// TIA Portal project "Boiler_KVGM20" (V14)
// Программа управления котлом КВГМ-20

(* hardware
DEVICE "ET 200SP station_1"  ET 200SP-Station
   slot 0: "Rack_0"  Rack  6ES5 710-8MAx1
   slot 1: "PLC_1"  CPU 1510SP-1 PN  6ES7 510-1DJ01-0AB0  V2.1
   slot 2: "AI 8xI 2-,4-wire BA_1"  AI 8xI 2-,4-wire BA  6ES7 134-6GF00-0AA1  V1.0
      slot 1: "AI 8xI 2-,4-wire BA_1"  AI 8xI 2-,4-wire BA
   slot 3: "AI 8xI 2-,4-wire BA_2"  AI 8xI 2-,4-wire BA  6ES7 134-6GF00-0AA1  V1.0
      slot 1: "AI 8xI 2-,4-wire BA_2"  AI 8xI 2-,4-wire BA
   slot 4: "AI 8xI 2-,4-wire BA_3"  AI 8xI 2-,4-wire BA  6ES7 134-6GF00-0AA1  V1.0
      slot 1: "AI 8xI 2-,4-wire BA_3"  AI 8xI 2-,4-wire BA
   slot 5: "DI 16x24VDC ST_1"  DI 16x24VDC ST  6ES7 131-6BH00-0BA0  V1.1
      slot 1: "DI 16x24VDC ST_1"  DI 16x24VDC ST
   slot 6: "DI 16x24VDC ST_2"  DI 16x24VDC ST  6ES7 131-6BH00-0BA0  V1.1
      slot 1: "DI 16x24VDC ST_2"  DI 16x24VDC ST
   slot 7: "DI 16x24VDC ST_3"  DI 16x24VDC ST  6ES7 131-6BH00-0BA0  V1.1
      slot 1: "DI 16x24VDC ST_3"  DI 16x24VDC ST
   slot 8: "DI 16x24VDC ST_4"  DI 16x24VDC ST  6ES7 131-6BH00-0BA0  V1.1
      slot 1: "DI 16x24VDC ST_4"  DI 16x24VDC ST
   slot 9: "DI 16x24VDC ST_5"  DI 16x24VDC ST  6ES7 131-6BH00-0BA0  V1.1
      slot 1: "DI 16x24VDC ST_5"  DI 16x24VDC ST
   slot 10: "DI 16x24VDC ST_6"  DI 16x24VDC ST  6ES7 131-6BH00-0BA0  V1.1
      slot 1: "DI 16x24VDC ST_6"  DI 16x24VDC ST
   slot 11: "DQ 16x24VDC/0.5A ST_1"  DQ 16x24VDC/0.5A ST  6ES7 132-6BH00-0BA0  V1.1
      slot 1: "DQ 16x24VDC/0.5A ST_1"  DQ 16x24VDC/0.5A ST
   slot 12: "DQ 16x24VDC/0.5A ST_2"  DQ 16x24VDC/0.5A ST  6ES7 132-6BH00-0BA0  V1.1
      slot 1: "DQ 16x24VDC/0.5A ST_2"  DQ 16x24VDC/0.5A ST
   slot 13: "DQ 16x24VDC/0.5A ST_3"  DQ 16x24VDC/0.5A ST  6ES7 132-6BH00-0BA0  V1.1
      slot 1: "DQ 16x24VDC/0.5A ST_3"  DQ 16x24VDC/0.5A ST
   slot 14: "AQ 4xU/I ST_1"  AQ 4xU/I ST  6ES7 135-6HD00-0BA1  V1.1
      slot 1: "AQ 4xU/I ST_1"  AQ 4xU/I ST
   slot 15: "Server module_1"  Server module  6ES7 193-6PA00-0AA0  V1.1
      slot 1: "Server module_1"  Server module
   slot 127: "BA 2xRJ45"  BA 2xRJ45  6ES7 193-6AR00-0AA0  V0.0
      slot 32769: "Port_1"  6ES7 193-6AR00-0AA0
      slot 32770: "Port_2"  6ES7 193-6AR00-0AA0
*)

// ===== PLC "PLC_1"  CPU 1510SP-1 PN =====

VAR_GLOBAL   // PLC tag table "Default tag table"
   "Module1Chanel1" AT %IW0 : Int;
   "Module1Chanel2" AT %IW2 : Int;
   "Module1Chanel3" AT %IW4 : Int;
   "Module1Chanel4" AT %IW6 : Int;
   "Module1Chanel5" AT %IW8 : Int;
   "Module1Chanel6" AT %IW10 : Int;
   "Module1Chanel7" AT %IW12 : Int;
   "Module1Chanel8" AT %IW14 : Int;
   "Module2Chanel1" AT %IW16 : Int;
   "Module2Chanel2" AT %IW18 : Int;
   "Module2Chanel3" AT %IW20 : Int;
   "Module2Chanel4" AT %IW22 : Int;
   "Module2Chanel5" AT %IW24 : Int;
   "Module2Chanel6" AT %IW26 : Int;
   "Module2Chanel7" AT %IW28 : Int;
   "Module2Chanel8" AT %IW30 : Int;
   "Module3Chanel1" AT %IW32 : Int;
   "Module3Chanel2" AT %IW34 : Int;
   "Module3Chanel3" AT %IW36 : Int;
   "Module3Chanel4" AT %IW38 : Int;
   "Module3Chanel5" AT %IW40 : Int;
   "Module3Chanel6" AT %IW42 : Int;
   "Module3Chanel7" AT %IW44 : Int;
   "Module3Chanel8" AT %IW46 : Int;
   "Module4Chanel1" AT %I48.0 : Bool;
   "Module4Chanel2" AT %I48.1 : Bool;
   "Module4Chanel3" AT %I48.2 : Bool;
   "Module4Chanel4" AT %I48.3 : Bool;
   "Module4Chanel5" AT %I48.4 : Bool;
   "Module4Chanel6" AT %I48.5 : Bool;
   "Module4Chanel7" AT %I48.6 : Bool;
   "Module4Chanel8" AT %I48.7 : Bool;
   "Module4Chanel9" AT %I49.0 : Bool;
   "Module4Chanel10" AT %I49.1 : Bool;
   "Module4Chanel11" AT %I49.2 : Bool;
   "Module4Chanel12" AT %I49.3 : Bool;
   "Module4Chanel13" AT %I49.4 : Bool;
   "Module4Chanel14" AT %I49.5 : Bool;
   "Module4Chanel15" AT %I49.6 : Bool;
   "Module4Chanel16" AT %I49.7 : Bool;
   "Module5Chanel1" AT %I50.0 : Bool;
   "Module5Chanel2" AT %I50.1 : Bool;
   "Module5Chanel3" AT %I50.2 : Bool;
   "Module5Chanel4" AT %I50.3 : Bool;
   "Module5Chanel5" AT %I50.4 : Bool;
   "Module5Chanel6" AT %I50.5 : Bool;
   "Module5Chanel7" AT %I50.6 : Bool;
   "Module5Chanel8" AT %I50.7 : Bool;
   "Module5Chanel9" AT %I51.0 : Bool;
   "Module5Chanel10" AT %I51.1 : Bool;
   "Module5Chanel11" AT %I51.2 : Bool;
   "Module5Chanel12" AT %I51.3 : Bool;
   "Module5Chanel13" AT %I51.4 : Bool;
   "Module5Chanel14" AT %I51.5 : Bool;
   "Module5Chanel15" AT %I51.6 : Bool;
   "Module5Chanel16" AT %I51.7 : Bool;
   "Module6Chanel1" AT %I52.0 : Bool;
   "Module6Chanel2" AT %I52.1 : Bool;
   "Module6Chanel3" AT %I52.2 : Bool;
   "Module6Chanel4" AT %I52.3 : Bool;
   "Module6Chanel5" AT %I52.4 : Bool;
   "Module6Chanel6" AT %I52.5 : Bool;
   "Module6Chanel7" AT %I52.6 : Bool;
   "Module6Chanel8" AT %I52.7 : Bool;
   "Module6Chanel9" AT %I53.0 : Bool;
   "Module6Chanel10" AT %I53.1 : Bool;
   "Module6Chanel11" AT %I53.2 : Bool;
   "Module6Chanel12" AT %I53.3 : Bool;
   "Module6Chanel13" AT %I53.4 : Bool;
   "Module6Chanel14" AT %I53.5 : Bool;
   "Module6Chanel15" AT %I53.6 : Bool;
   "Module6Chanel16" AT %I53.7 : Bool;
   "Module7Chanel1" AT %I54.0 : Bool;
   "Module7Chanel2" AT %I54.1 : Bool;
   "Module7Chanel3" AT %I54.2 : Bool;
   "Module7Chanel4" AT %I54.3 : Bool;
   "Module7Chanel5" AT %I54.4 : Bool;
   "Module7Chanel6" AT %I54.5 : Bool;
   "Module7Chanel7" AT %I54.6 : Bool;
   "Module7Chanel8" AT %I54.7 : Bool;
   "Module7Chanel9" AT %I55.0 : Bool;
   "Module7Chanel10" AT %I55.1 : Bool;
   "Module7Chanel11" AT %I55.2 : Bool;
   "Module7Chanel12" AT %I55.3 : Bool;
   "Module7Chanel13" AT %I55.4 : Bool;
   "Module7Chanel14" AT %I55.5 : Bool;
   "Module7Chanel15" AT %I55.6 : Bool;
   "Module7Chanel16" AT %I55.7 : Bool;
   "Module8Chanel1" AT %I56.0 : Bool;
   "Module8Chanel2" AT %I56.1 : Bool;
   "Module8Chanel3" AT %I56.2 : Bool;
   "Module8Chanel4" AT %I56.3 : Bool;
   "Module8Chanel5" AT %I56.4 : Bool;
   "Module8Chanel6" AT %I56.5 : Bool;
   "Module8Chanel7" AT %I56.6 : Bool;
   "Module8Chanel8" AT %I56.7 : Bool;
   "Module8Chanel9" AT %I57.0 : Bool;
   "Module8Chanel10" AT %I57.1 : Bool;
   "Module8Chanel11" AT %I57.2 : Bool;
   "Module8Chanel12" AT %I57.3 : Bool;
   "Module8Chanel13" AT %I57.4 : Bool;
   "Module8Chanel14" AT %I57.5 : Bool;
   "Module8Chanel15" AT %I57.6 : Bool;
   "Module8Chanel16" AT %I57.7 : Bool;
   "Module9Chanel1" AT %I58.0 : Bool;
   "Module9Chanel2" AT %I58.1 : Bool;
   "Module9Chanel3" AT %I58.2 : Bool;
   "Module9Chanel4" AT %I58.3 : Bool;
   "Module9Chanel5" AT %I58.4 : Bool;
   "Module9Chanel6" AT %I58.5 : Bool;
   "Module9Chanel7" AT %I58.6 : Bool;
   "Module9Chanel8" AT %I58.7 : Bool;
   "Module9Chanel9" AT %I59.0 : Bool;
   "Module9Chanel10" AT %I59.1 : Bool;
   "Module9Chanel11" AT %I59.2 : Bool;
   "Module9Chanel12" AT %I59.3 : Bool;
   "Module9Chanel13" AT %I59.4 : Bool;
   "Module9Chanel14" AT %I59.5 : Bool;
   "Module9Chanel15" AT %I59.6 : Bool;
   "Module9Chanel16" AT %I59.7 : Bool;
   "Module10Chanel1" AT %Q0.0 : Bool;
   "Module10Chanel8" AT %Q0.7 : Bool;
   "Module10Chanel7" AT %Q0.6 : Bool;
   "Module10Chanel6" AT %Q0.5 : Bool;
   "Module10Chanel5" AT %Q0.4 : Bool;
   "Module10Chanel4" AT %Q0.3 : Bool;
   "Module10Chanel3" AT %Q0.2 : Bool;
   "Module10Chanel2" AT %Q0.1 : Bool;
   "Module10Chanel9" AT %Q1.0 : Bool;
   "Module10Chanel10" AT %Q1.1 : Bool;
   "Module10Chanel11" AT %Q1.2 : Bool;
   "Module10Chanel12" AT %Q1.3 : Bool;
   "Module10Chanel13" AT %Q1.4 : Bool;
   "Module10Chanel14" AT %Q1.5 : Bool;
   "Module10Chanel15" AT %Q1.6 : Bool;
   "Module10Chanel16" AT %Q1.7 : Bool;
   "Module11Chanel1" AT %Q2.0 : Bool;
   "Module11Chanel2" AT %Q2.1 : Bool;
   "Module11Chanel3" AT %Q2.2 : Bool;
   "Module11Chanel4" AT %Q2.3 : Bool;
   "Module11Chanel5" AT %Q2.4 : Bool;
   "Module11Chanel6" AT %Q2.5 : Bool;
   "Module11Chanel7" AT %Q2.6 : Bool;
   "Module11Chanel8" AT %Q2.7 : Bool;
   "Module11Chanel9" AT %Q3.0 : Bool;
   "Module11Chanel10" AT %Q3.1 : Bool;
   "Module11Chanel11" AT %Q3.2 : Bool;
   "Module11Chanel12" AT %Q3.3 : Bool;
   "Module11Chanel13" AT %Q3.4 : Bool;
   "Module11Chanel14" AT %Q3.5 : Bool;
   "Module11Chanel15" AT %Q3.6 : Bool;
   "Module11Chanel16" AT %Q3.7 : Bool;
   "Module12Chanel1" AT %Q4.0 : Bool;
   "Module12Chanel2" AT %Q4.1 : Bool;
   "Module12Chanel3" AT %Q4.2 : Bool;
   "Module12Chanel4" AT %Q4.3 : Bool;
   "Module12Chanel5" AT %Q4.4 : Bool;
   "Module12Chanel6" AT %Q4.5 : Bool;
   "Module12Chanel7" AT %Q4.6 : Bool;
   "Module12Chanel8" AT %Q4.7 : Bool;
   "Module12Chanel9" AT %Q5.0 : Bool;
   "Module12Chanel10" AT %Q5.1 : Bool;
   "Module12Chanel11" AT %Q5.2 : Bool;
   "Module12Chanel12" AT %Q5.3 : Bool;
   "Module12Chanel13" AT %Q5.4 : Bool;
   "Module12Chanel14" AT %Q5.5 : Bool;
   "Module12Chanel15" AT %Q5.6 : Bool;
   "Module12Chanel16" AT %Q5.7 : Bool;
   "Module13Chanel1" AT %QW6 : Int;
   "Module13Chanel2" AT %QW8 : Int;
   "Module13Chanel3" AT %QW10 : Int;
   "Module13Chanel4" AT %QW12 : Int;
   "FRONT_Btn_Ventilation_HMI" AT %M9.2 : Bool;   // Фронт нажатия кнопки ВЕНТИЛЯЦИЯ на HMI
   "FRONT_Btn_Ventilation_SCADA" AT %M9.3 : Bool;   // Фронт нажатия кнопки ВЕНТИЛЯЦИЯ на SCADA
   "FRONT_Btn_Ignition_HMI" AT %M9.4 : Bool;   // Фронт нажатия кнопки РОЗЖИГ на HMI
   "FRONT_Btn_Ignition_SCADA" AT %M9.5 : Bool;   // Фронт нажатия кнопки РОЗЖИГ на SCADA
   "FRONT_Btn_Normal_stop_HMI" AT %M9.6 : Bool;   // Фронт нажатия кнопки НОРМАЛЬНЫЙ ОСТАНОВ на HMI
   "FRONT_Btn_Normal_stop_SCADA" AT %M9.7 : Bool;   // Фронт нажатия кнопки НОРМАЛЬНЫЙ ОСТАНОВ на SCADA
   "FRONT_Btn_Alarm_stop_HMI" AT %M10.0 : Bool;   // Фронт нажатия кнопки АВАРИЙНЫЙ ОСТАНОВ на HMI
   "FRONT_Btn_Alarm_stop_SCADA" AT %M10.1 : Bool;   // Фронт нажатия кнопки АВАРИЙНЫЙ ОСТАНОВ на SCADA
   "FRONT_Btn_test_press_HMI" AT %M10.2 : Bool;   // Фронт нажатия кнопки ТЕСТОВАЯ ОПРЕССОВКА на HMI
   "FRONT_Btn_test_ignition_HMI" AT %M10.3 : Bool;   // Фронт нажатия кнопки ТЕСТОВЫЙ РОЗЖИГ на HMI
   "FRONT_Btn_manual_ignition_HMI" AT %M10.4 : Bool;   // Фронт нажатия кнопки РУЧНОЙ РОЗЖИГ на HMI
   "Gen_imp" AT %M10.5 : Bool;
   "FRONT_Alarm_1" AT %M10.6 : Bool;   // Фронт аварии1
   "FRONT_Alarm_2" AT %M10.7 : Bool;   // Фронт аварии2
   "FRONT_Alarm_3" AT %M11.0 : Bool;   // Фронт аварии3
   "FRONT_Alarm_4" AT %M11.1 : Bool;   // Фронт аварии4
   "FRONT_Alarm_5" AT %M11.2 : Bool;   // Фронт аварии5
   "FRONT_Alarm_6" AT %M11.3 : Bool;   // Фронт аварии6
   "FRONT_Alarm_7" AT %M11.4 : Bool;   // Фронт аварии7
   "FRONT_Alarm_8" AT %M11.5 : Bool;   // Фронт аварии8
   "FRONT_Alarm_9" AT %M11.6 : Bool;   // Фронт аварии9
   "FRONT_Alarm_10" AT %M11.7 : Bool;   // Фронт аварии10
   "FRONT_Alarm_11" AT %M12.0 : Bool;   // Фронт аварии11
   "FRONT_Alarm_12" AT %M12.1 : Bool;   // Фронт аварии12
   "FRONT_Alarm_13" AT %M12.2 : Bool;   // Фронт аварии13
   "FRONT_Alarm_14" AT %M12.3 : Bool;   // Фронт аварии14
   "FRONT_Alarm_15" AT %M12.4 : Bool;   // Фронт аварии15
   "FRONT_Alarm_16" AT %M12.5 : Bool;   // Фронт аварии16
   "FRONT_Alarm_17" AT %M12.6 : Bool;   // Фронт аварии17
   "FRONT_Btn_reset_sound_HMI" AT %M12.7 : Bool;   // Фронт нажатия кнопки СБРОС ЗВУКА на HMI
   "FRONT_DS_mode" AT %M13.0 : Bool;   // Фронт перевода ДС в ручной режим
   "FRONT_DV_mode" AT %M13.1 : Bool;   // Фронт перевода ДВ в ручной режим
   "FRONT_IVN_mode" AT %M13.2 : Bool;   // Фронт перевода ИВН в ручной режим
   "FRONT_KB_mode" AT %M13.3 : Bool;   // Фронт перевода КБ в ручной режим
   "FRONT_KO_mode" AT %M13.4 : Bool;   // Фронт перевода КО в ручной режим
   "FRONT_KZ_mode" AT %M13.5 : Bool;   // Фронт перевода КЗ в ручной режим
   "FRONT_PZK1_mode" AT %M13.6 : Bool;   // Фронт перевода ПЗК1 в ручной режим
   "FRONT_PZK2_mode" AT %M13.7 : Bool;   // Фронт перевода ПЗК2 в ручной режим
END_VAR

VAR_GLOBAL   // PLC tag table "www"
   "retval" AT %IW60 : Int;
END_VAR

TYPE "AI_sensor_4_20"
   STRUCT
      Enable : Bool;   // Наличие датчика
      N_module : USInt;   // № модуля (начиная с 1)
      N_chanel : USInt;   // № канала (начиная с 1)
      Value : Real;   // Текущее значение в физической величине
      Current_ADC : Int;   // Текущий код АЦП
      Low_limit_phisical_current : Real;   // Нижний предел датчика в физической величине текущий
      High_limit_phisical_current : Real := 100.0;   // Верхний предел датчика в физической величине текущий
      Low_limit_ADC_current : Int;   // Нижний предел датчика в АЦП текущий
      High_limit_ADC_current : Int := 27648;   // Верхний предел датчика в АЦП текущий
      Low_limit_phisical_new : Real;   // Нижний предел датчика в физической величине новый
      High_limit_phisical_new : Real := 100.0;   // Верхний предел датчика в физической величине новый
      Low_limit_ADC_new : Int;   // Нижний предел датчика в АЦП новый
      High_limit_ADC_new : Int := 27648;   // Верхний предел датчика в АЦП новый
      Apply : Bool;   // Применить
      Alarm_sensor : Bool;   // Неисправность датчика
      Current : Real;   // Текущее значение тока
      Reserv1 : Real;
      Reserv2 : Real;
      Reserv3 : Real;
      Reserv4 : Real;
   END_STRUCT;
END_TYPE

TYPE "DI_sensor"
   STRUCT
      Enable : Bool;   // Наличие датчика
      N_module : USInt;   // № модуля (начиная с 4)
      N_chanel : USInt;   // № канала (начиная с 1)
      Invert : Bool;   // Необходимость инвертирования сигнала
      Value : Bool;   // Текущее значение сигнала
      reserv1 : Bool;
      reserv2 : Bool;
   END_STRUCT;
END_TYPE

TYPE "DO_signal"
   STRUCT
      Enable : Bool;   // Наличие сигнала
      N_module : USInt;   // № модуля (начиная с 10)
      N_chanel : USInt;   // № канала (начиная с 1)
      Value : Bool;   // Текущее значение сигнала
      reserv1 : Bool;
      reserv2 : Bool;
   END_STRUCT;
END_TYPE

TYPE "AO_signal"
   STRUCT
      Enable : Bool;   // Наличие датчика
      N_module : USInt;   // № модуля (начиная с 13)
      N_chanel : USInt;   // № канала (начиная с 1)
      Value : Real;   // Текущее значение в физической величине
      Current_DAC : Int;   // Текущий код ЦАП
      Low_limit_phisical_current : Real;   // Нижний предел датчика в физической величине текущий
      High_limit_phisical_current : Real := 100.0;   // Верхний предел датчика в физической величине текущий
      Low_limit_phisical_new : Real;   // Нижний предел датчика в физической величине новый
      High_limit_phisical_new : Real := 100.0;   // Верхний предел датчика в физической величине новый
      Apply : Bool;   // Применить
      Reserv1 : Real;
      Reserv2 : Real;
      Reserv3 : Real;
      Reserv4 : Real;
   END_STRUCT;
END_TYPE

TYPE "Q_water"
   STRUCT
      Enable : Bool;   // Наличие параметра
      Value : Real;   // Значение
      "a" : Real := 0.6038;   // Коэффициент расхода
      Ksh : Real := 1.0;   // Поправочный коэффициент на шероховатость трубопровода
      Kp : Real := 1.00409;   // Поправочный коэффициент на неостроту входной кромки диафрагмы
      d : Real := 0.070696;   // Диаметр сужающего устройства
      ro : Real := 962.4729;   // Плотность среды в рабочих условиях
   END_STRUCT;
END_TYPE

TYPE "Q_gas"
   STRUCT
      Enable : Bool;   // Наличие параметра
      Value : Real;   // Значение
      "a" : Real := 0.60631;   // Коэффициент расхода
      Ksh : Real := 1.0;   // Поправочный коэффициент на шероховатость трубопровода
      Kp : Real := 1.00373;   // Поправочный коэффициент на неостроту входной кромки диафрагмы
      "E" : Real;   // Коэффициент расширения
      d : Real := 0.075498;   // Диаметр сужающего устройства
      ros : Real := 0.67245;   // Плотность среды в стандартных условиях
      Ps : Real := 101325.0;   // Давление в нормальных условиях
      Tgas : Real;   // Температура газа в рабочих условиях
      Tgas_fixed_value : Real;   // Температура газа в рабочих условиях фиксированное значение
      Tgas_fixed_value_on : Bool;   // Температура газа в рабочих условиях включить фиксированное значение
      K : Real := 0.99832;   // Коэффициент сжимаемости
      B4 : Real;   // Относительный диаметр сужающего устройства (в 4 степени)
      Dtrub : Real := 0.207;   // Диаметр трубопровода
      Pgas : Real;   // Давление газа в рабочих условиях
      Pgas_fixed_value : Real;   // Давление газа в рабочих условиях фиксированное значение
      Pgas_fixed_value_on : Bool;   // Давление газа в рабочих условиях включить фиксированное значение
   END_STRUCT;
END_TYPE

DATA_BLOCK "Sensors"   // DB1
{ S7_Optimized_Access := 'FALSE' }
VERSION : 0.1
   VAR
      T_water_before_boiler : "AI_sensor_4_20";   // Температура сетевой воды перед котлом (град С)
      P_water_before_boiler : "AI_sensor_4_20";   // Давление сетевой воды перед котлом (кгс/см2)
      dP_water_boiler : "AI_sensor_4_20";   // Перепад давления сетевой воды через котел (кПа)
      T_water_after_boiler : "AI_sensor_4_20";   // Температура сетевой воды после котла (град С)
      P_water_after_boiler : "AI_sensor_4_20";   // Давление сетевой воды после котла (кгс/см2)
      dP_water_boiler_1 : "AI_sensor_4_20";   // Перепад давления сетевой воды через котел (кПа)
      P_water_before_boiler_1 : "AI_sensor_4_20";   // Давление сетевой воды перед котлом (кгс/см2)
      dP_gas_boiler : "AI_sensor_4_20";   // Перепад давления газа на котел (кПа)
      dP_furnace_boiler : "AI_sensor_4_20";   // Разрежение в топке котла (Па)
      P_gas_before_PZK1_and_PZK2 : "AI_sensor_4_20";   // Давление газа между ПЗК-1 и ПЗК-2 (кПа)
      P_gas_before_burner : "AI_sensor_4_20";   // Давление газа перед горелкой (кПа)
      P_air_burner : "AI_sensor_4_20";   // Давление воздуха к горелке (Па)
      T_exhaust_gas : "AI_sensor_4_20";   // Температура уходящих газов (град С)
      ZRG_position : "AI_sensor_4_20";   // Положение рег. заслонки газа перед котлом (%)
      NAV_position : "AI_sensor_4_20";   // Положение направл. аппарата вентилятора (%)
      NAD_position : "AI_sensor_4_20";   // Положение направл. аппарата дымососа (%)
      DV_current_frequency : "AI_sensor_4_20";   // Текущ. значение ПЧ ДВ (Гц)
      DS_current_frequency : "AI_sensor_4_20";   // Текущ. значение ПЧ ДС (Гц)
      T_gas_before_BG : "AI_sensor_4_20";   // Температура газа перед БГ (град С)
      P_gas_before_BG : "AI_sensor_4_20";   // Давление газа перед БГ (кПа)
      Burner_flame : "DI_sensor";   // Наличие пламени горелки
      Igniter_flame : "DI_sensor";   // Наличие пламени запальника горелки
      KB_close : "DI_sensor";   // Клапан безопасности закрыт
      KO_open : "DI_sensor";   // Клапан опрессовки открыт
      KZ_open : "DI_sensor";   // Клапан запальника открыт
      PZK1_open : "DI_sensor";   // ПЗК-1 горелки открыт
      PZK2_not_close : "DI_sensor";   // ПЗК-2 горелки не закрыт
      P_gas_before_BG_min : "DI_sensor";   // Давление газа перед БГ мин.
      P_gas_before_BG_max : "DI_sensor";   // Давление газа перед БГ макс.
      P_air_before_burner_min : "DI_sensor";   // Давление воздуха перед горелкой мин.
      P_gas_before_burner_min : "DI_sensor";   // Давление газа перед горелкой мин.
      P_gas_before_burner_max : "DI_sensor";   // Давление газа перед горелкой макс.
      ZRG_open : "DI_sensor";   // Регулирующая заслонка газа. открыта
      ZRG_close : "DI_sensor";   // Регулирующая заслонка газа. закрыта
      ZRG_middle : "DI_sensor";   // Регулирующая заслонка газа. среднее
      ZRG_avto : "DI_sensor";   // Регулирующая заслонка газа. БРУ в положении "Авт"
      NAV_open : "DI_sensor";   // Регулирующая заслонка НАВ. открыта
      NAV_close : "DI_sensor";   // Регулирующая заслонка НАВ. закрыта
      NAV_middle : "DI_sensor";   // Регулирующая заслонка НАВ. среднее
      NAV_avto : "DI_sensor";   // Регулирующая заслонка НАВ. БРУ в положении "Авт"
      NAD_open : "DI_sensor";   // Регулирующая заслонка НАД. открыта
      NAD_close : "DI_sensor";   // Регулирующая заслонка НАД. закрыта
      NAD_middle : "DI_sensor";   // Регулирующая заслонка НАД. среднее
      NAD_avto : "DI_sensor";   // Регулирующая заслонка НАД. БРУ в положении "Авт"
      dP_furnace_boiler_min : "DI_sensor";   // Разрежение в топке котла мин.
      T_water_after_boiler_max : "DI_sensor";   // Температура сетевой воды после котла макс.
      Q_water_boiler_min : "DI_sensor";   // Расход сетевой воды через котел мин.
      Q_water_boiler_max : "DI_sensor";   // Расход сетевой воды через котел макс.
      P_water_after_boiler_min : "DI_sensor";   // Давление сетевой воды после котла мин.
      P_water_after_boiler_max : "DI_sensor";   // Давление сетевой воды после котла макс.
      P_water_before_boiler_min : "DI_sensor";   // Давление сетевой воды перед котлом мин.
      P_water_before_boiler_max : "DI_sensor";   // Давление сетевой воды перед котлом макс.
      Call_power_supply_сabinet : "DI_sensor";   // Вызов к шакафу электропитания
      DV_Invertor_alarm : "DI_sensor";   // Авария ПЧ ДВ
      DV_local_control : "DI_sensor";   // Управление «Местный» ДВ
      DV_dist_control : "DI_sensor";   // Управление «Дистанционный» ДВ
      DV_powergrid_mode : "DI_sensor";   // Режим "СЕТЬ" ДВ
      DV_invertor_mode : "DI_sensor";   // Режим "ПЧ" ДВ
      DV_invertor_QF_on : "DI_sensor";   // Автомат работы ДВ от ПЧ включен
      DV_powergrid_QF_on : "DI_sensor";   // Автомат работы ДВ от сети включен
      DV_invertor_on : "DI_sensor";   // Включен ДВ от ПЧ
      DV_powergrid_on : "DI_sensor";   // Включен ДВ от сети
      DV_no_voltage : "DI_sensor";   // Нет напряжения сети ШУД ДВ
      DS_Invertor_alarm : "DI_sensor";   // Авария ПЧ ДС
      DS_local_control : "DI_sensor";   // Управление «Местный» ДС
      DS_dist_control : "DI_sensor";   // Управление «Дистанционный» ДС
      DS_powergrid_mode : "DI_sensor";   // Режим "СЕТЬ" ДС
      DS_invertor_mode : "DI_sensor";   // Режим "ПЧ" ДС
      DS_invertor_QF_on : "DI_sensor";   // Автомат работы ДС от ПЧ включен
      DS_powergrid_QF_on : "DI_sensor";   // Автомат работы ДС от сети включен
      DS_invertor_on : "DI_sensor";   // ДС включен от ПЧ
      DS_powergrid_on : "DI_sensor";   // ДС включен от сети
      DS_no_voltage : "DI_sensor";   // Нет напряжения сети ШУД ДС
      CO_1 : "DI_sensor";   // Загазованность СО I порог
      CO_2 : "DI_sensor";   // Загазованность СО II порог
      CH4 : "DI_sensor";   // Загазованность CH4 порог
      Btn_STOP : "DI_sensor";   // Кнопка СТОП
      Btn_Ventilation : "DI_sensor";   // Кнопка Вентиляция
      Btn_Ignition : "DI_sensor";   // Кнопка Розжиг
      Btn_Sound : "DI_sensor";   // Кнопка Сброс звука / Проверка звука
      SHEU_voltage_ok : "DI_sensor";   // Контроль питания сети ~400В 1ШЭУ
      PZK2_open : "DI_sensor";   // ПЗК-2 горелки открыт
      Power_PLC_from_UPS : "DI_sensor";   // Питание контроллера от ИБП
      UPS_Low_charge : "DI_sensor";   // Заряд батареи ИБП низкий
      ZRG_voltage_ok : "DI_sensor";   // ЗРГ Напряжение в норме
      NAV_voltage_ok : "DI_sensor";   // НАВ Напряжение в норме
      NAD_voltage_ok : "DI_sensor";   // НАД Напряжение в норме
      ZDG_no_open : "DI_sensor";   // ЗДГ перед БГ. не открыта
      ZDG_no_close : "DI_sensor";   // ЗДГ перед БГ. не закрыта
      ZDG_opening : "DI_sensor";   // ЗДГ перед БГ. ход открытие
      ZDG_closing : "DI_sensor";   // ЗДГ перед БГ. ход закрытие
      ZDG_voltage_ok : "DI_sensor";   // ЗДГ перед БГ. Напряжение в норме
      ZDSV_before_boiler_no_open : "DI_sensor";   // ЗДСВ перед котлом. не открыта
      ZDSV_before_boiler_no_close : "DI_sensor";   // ЗДСВ перед котлом. не закрыта
      ZDSV_before_boiler_opening : "DI_sensor";   // ЗДСВ перед котлом. ход открытие
      ZDSV_before_boiler_closing : "DI_sensor";   // ЗДСВ перед котлом. ход закрытие
      ZDSV_before_boiler_voltage_ok : "DI_sensor";   // ЗДСВ перед котлом. Напряжение в норме
      ZDSV_before_boiler_limit_rotational_moment : "DI_sensor";   // ЗДСВ перед котлом. ограничитель крутящего момента
      ZDSV_after_boiler_no_open : "DI_sensor";   // ЗДСВ после котла. не открыта
      ZDSV_after_boiler_no_close : "DI_sensor";   // ЗДСВ после котла. не закрыта
      ZDSV_after_boiler_opening : "DI_sensor";   // ЗДСВ после котла. ход открытие
      ZDSV_after_boiler_closing : "DI_sensor";   // ЗДСВ после котла. ход закрытие
      ZDSV_after_boiler_voltage_ok : "DI_sensor";   // ЗДСВ после котла. Напряжение в норме
      ZDSV_after_boiler_limit_rotational_moment : "DI_sensor";   // ЗДСВ после котла. ограничитель крутящего момента
      ZRG_control_open : "DO_signal";   // ЗРГ команда «Больше»
      ZRG_control_close : "DO_signal";   // ЗРГ команда «Меньше»
      NAV_control_open : "DO_signal";   // НАВ команда «Больше»
      NAV_control_close : "DO_signal";   // НАВ команда «Меньше»
      NAD_control_open : "DO_signal";   // НАД команда «Больше»
      NAD_control_close : "DO_signal";   // НАД команда «Меньше»
      Indication_RUN : "DO_signal";   // Индикация «Работа»
      Indication_ALARM : "DO_signal";   // Индикация «Авария»
      Indication_NORMA : "DO_signal";   // Индикация «Защиты в норме»
      Indication_READY : "DO_signal";   // Индикация «Готов к розжигу»
      ZDG_control_open : "DO_signal";   // ЗДГ команда «открыть»
      ZDG_control_close : "DO_signal";   // ЗДГ команда «закрыть»
      ZDG_control_stop : "DO_signal";   // ЗДГ команда «стоп»
      ZDG_control_disable_open : "DO_signal";   // ЗДГ команда «запрет открытия»
      KB_control_close : "DO_signal";   // КБ команда «закрыть»
      KO_control_open : "DO_signal";   // КО команда «открыть»
      KZ_control_open : "DO_signal";   // КЗ команда «открыть»
      IVN_control_on : "DO_signal";   // ИВН команда «включить»
      PZK1_control_open : "DO_signal";   // ПЗК1 команда «открыть»
      PZK2_control_open : "DO_signal";   // ПЗК2 команда «открыть»
      ZDSV_before_boiler_control_open : "DO_signal";   // ЗДСВ перед котлом команда «открыть»
      ZDSV_before_boiler_control_close : "DO_signal";   // ЗДСВ перед котлом команда «закрыть»
      ZDSV_before_boiler_control_stop : "DO_signal";   // ЗДСВ перед котлом команда «стоп»
      ZDSV_before_boiler_control_disable_close : "DO_signal";   // ЗДСВ перед котлом команда «запрет закрытия»
      ZDSV_after_boiler_control_open : "DO_signal";   // ЗДСВ после котла команда «открыть»
      ZDSV_after_boiler_control_close : "DO_signal";   // ЗДСВ после котла команда «закрыть»
      ZDSV_after_boiler_control_stop : "DO_signal";   // ЗДСВ после котла команда «стоп»
      ZDSV_after_boiler_control_disable_close : "DO_signal";   // ЗДСВ после котла команда «запрет закрытия»
      control_alarm_signal : "DO_signal";   // Включение аварийной сигнализации
      DV_control_start : "DO_signal";   // ДВ команда «пуск»
      DV_control_stop : "DO_signal";   // ДВ команда «стоп»
      DS_control_start : "DO_signal";   // ДС команда «пуск»
      DS_control_stop : "DO_signal";   // ДС команда «стоп»
      DV_control_frequency : "AO_signal";   // Задание для ПЧ ДВ
      DS_control_frequency : "AO_signal";   // Задание для ПЧ ДС
      Q_water_boiler : "Q_water";   // Расход сетевой воды через котел (м3/ч)
      Q_gas : "Q_gas";   // Расход газа (м3/ч)
   END_VAR
BEGIN
   T_water_before_boiler.Enable := true;
   T_water_before_boiler.N_module := 1;
   T_water_before_boiler.N_chanel := 1;
   P_water_before_boiler.Enable := true;
   dP_water_boiler.Enable := true;
   T_water_after_boiler.Enable := true;
   P_water_after_boiler.Enable := true;
   dP_water_boiler_1.Enable := true;
   P_water_before_boiler_1.Enable := true;
   dP_gas_boiler.Enable := true;
   dP_furnace_boiler.Enable := true;
   P_gas_before_PZK1_and_PZK2.Enable := true;
   P_gas_before_burner.Enable := true;
   P_air_burner.Enable := true;
   T_exhaust_gas.Enable := true;
   ZRG_position.Enable := true;
   NAV_position.Enable := true;
   NAD_position.Enable := true;
   DV_current_frequency.Enable := true;
   DS_current_frequency.Enable := true;
   P_water_before_boiler.N_module := 1;
   P_water_before_boiler.N_chanel := 2;
   dP_water_boiler.N_module := 1;
   dP_water_boiler.N_chanel := 3;
   T_water_after_boiler.N_module := 1;
   T_water_after_boiler.N_chanel := 4;
   P_water_after_boiler.N_module := 1;
   P_water_after_boiler.N_chanel := 5;
   dP_water_boiler_1.N_module := 1;
   dP_water_boiler_1.N_chanel := 6;
   P_water_before_boiler_1.N_module := 1;
   P_water_before_boiler_1.N_chanel := 7;
   dP_gas_boiler.N_module := 1;
   dP_gas_boiler.N_chanel := 8;
   dP_furnace_boiler.N_module := 2;
   dP_furnace_boiler.N_chanel := 1;
   P_gas_before_PZK1_and_PZK2.N_module := 2;
   P_gas_before_PZK1_and_PZK2.N_chanel := 2;
   P_gas_before_burner.N_module := 2;
   P_gas_before_burner.N_chanel := 3;
   P_air_burner.N_module := 2;
   P_air_burner.N_chanel := 4;
   T_exhaust_gas.N_module := 2;
   T_exhaust_gas.N_chanel := 5;
   ZRG_position.N_module := 2;
   ZRG_position.N_chanel := 6;
   NAV_position.N_module := 2;
   NAV_position.N_chanel := 7;
   NAD_position.N_module := 2;
   NAD_position.N_chanel := 8;
   DV_current_frequency.N_module := 3;
   DV_current_frequency.N_chanel := 1;
   DS_current_frequency.N_module := 3;
   DS_current_frequency.N_chanel := 2;
   T_water_before_boiler.Low_limit_phisical_current := 0.0;
   T_water_before_boiler.High_limit_phisical_current := 200.0;
   T_water_before_boiler.Low_limit_phisical_new := 0.0;
   T_water_before_boiler.High_limit_phisical_new := 200.0;
   dP_gas_boiler.High_limit_phisical_current := 16.0;
   dP_gas_boiler.High_limit_phisical_new := 16.0;
   P_gas_before_PZK1_and_PZK2.High_limit_phisical_current := 40.0;
   P_gas_before_PZK1_and_PZK2.High_limit_phisical_new := 40.0;
   P_gas_before_burner.High_limit_phisical_current := 40.0;
   P_gas_before_burner.High_limit_phisical_new := 40.0;
   dP_furnace_boiler.Low_limit_phisical_current := -200.0;
   dP_furnace_boiler.High_limit_phisical_current := 200.0;
   dP_furnace_boiler.Low_limit_phisical_new := -200.0;
   dP_furnace_boiler.High_limit_phisical_new := 200.0;
   T_exhaust_gas.High_limit_phisical_current := 300.0;
   T_exhaust_gas.High_limit_phisical_new := 300.0;
   P_air_burner.High_limit_phisical_current := 2500.0;
   P_air_burner.High_limit_phisical_new := 2500.0;
   T_water_after_boiler.High_limit_phisical_current := 200.0;
   T_water_after_boiler.High_limit_phisical_new := 200.0;
   P_water_before_boiler.High_limit_phisical_current := 160.0;
   P_water_before_boiler.High_limit_phisical_new := 160.0;
   dP_water_boiler.High_limit_phisical_current := 400.0;
   dP_water_boiler.High_limit_phisical_new := 400.0;
   P_water_after_boiler.High_limit_phisical_current := 16.0;
   P_water_after_boiler.High_limit_phisical_new := 16.0;
   dP_water_boiler_1.High_limit_phisical_current := 400.0;
   dP_water_boiler_1.High_limit_phisical_new := 400.0;
   P_water_before_boiler_1.High_limit_phisical_new := 16.0;
   P_water_before_boiler_1.High_limit_phisical_current := 16.0;
   DV_current_frequency.High_limit_phisical_current := 50.0;
   DV_current_frequency.High_limit_phisical_new := 50.0;
   DS_current_frequency.High_limit_phisical_current := 50.0;
   DS_current_frequency.High_limit_phisical_new := 50.0;
   T_gas_before_BG.High_limit_phisical_current := 200.0;
   T_gas_before_BG.High_limit_phisical_new := 200.0;
   P_gas_before_BG.High_limit_phisical_current := 40.0;
   P_gas_before_BG.High_limit_phisical_new := 40.0;
   Burner_flame.Enable := true;
   Igniter_flame.Enable := true;
   KB_close.Enable := true;
   KO_open.Enable := true;
   KZ_open.Enable := true;
   PZK1_open.Enable := true;
   PZK2_not_close.Enable := true;
   P_gas_before_BG_min.Enable := true;
   P_gas_before_BG_max.Enable := true;
   P_air_before_burner_min.Enable := true;
   P_gas_before_burner_min.Enable := true;
   P_gas_before_burner_max.Enable := true;
   ZRG_open.Enable := true;
   ZRG_close.Enable := true;
   ZRG_middle.Enable := true;
   ZRG_avto.Enable := true;
   NAV_open.Enable := true;
   NAV_close.Enable := true;
   NAV_middle.Enable := true;
   NAV_avto.Enable := true;
   NAD_open.Enable := true;
   NAD_close.Enable := true;
   NAD_middle.Enable := true;
   NAD_avto.Enable := true;
   dP_furnace_boiler_min.Enable := true;
   T_water_after_boiler_max.Enable := true;
   Q_water_boiler_min.Enable := true;
   Q_water_boiler_max.Enable := true;
   P_water_after_boiler_min.Enable := true;
   P_water_after_boiler_max.Enable := true;
   P_water_before_boiler_min.Enable := true;
   P_water_before_boiler_max.Enable := true;
   Call_power_supply_сabinet.Enable := true;
   DV_Invertor_alarm.Enable := true;
   DV_local_control.Enable := true;
   DV_dist_control.Enable := true;
   DV_powergrid_mode.Enable := true;
   DV_invertor_mode.Enable := true;
   DV_invertor_QF_on.Enable := true;
   DV_powergrid_QF_on.Enable := true;
   DV_invertor_on.Enable := true;
   DV_powergrid_on.Enable := true;
   DV_no_voltage.Enable := true;
   DS_Invertor_alarm.Enable := true;
   DS_local_control.Enable := true;
   DS_dist_control.Enable := true;
   DS_powergrid_mode.Enable := true;
   DS_invertor_mode.Enable := true;
   DS_invertor_QF_on.Enable := true;
   DS_powergrid_QF_on.Enable := true;
   DS_invertor_on.Enable := true;
   DS_powergrid_on.Enable := true;
   DS_no_voltage.Enable := true;
   CO_1.Enable := true;
   CO_2.Enable := true;
   CH4.Enable := true;
   SHEU_voltage_ok.Enable := true;
   PZK2_open.Enable := true;
   Power_PLC_from_UPS.Enable := true;
   ZRG_voltage_ok.Enable := true;
   NAV_voltage_ok.Enable := true;
   NAD_voltage_ok.Enable := true;
   ZDG_no_open.Enable := true;
   ZDG_no_close.Enable := true;
   ZDG_opening.Enable := true;
   ZDG_closing.Enable := true;
   ZDG_voltage_ok.Enable := true;
   ZDSV_before_boiler_no_open.Enable := true;
   ZDSV_before_boiler_no_close.Enable := true;
   ZDSV_before_boiler_opening.Enable := true;
   ZDSV_before_boiler_closing.Enable := true;
   ZDSV_before_boiler_voltage_ok.Enable := true;
   ZDSV_before_boiler_limit_rotational_moment.Enable := true;
   ZDSV_after_boiler_no_open.Enable := true;
   ZDSV_after_boiler_no_close.Enable := true;
   ZDSV_after_boiler_opening.Enable := true;
   ZDSV_after_boiler_closing.Enable := true;
   ZDSV_after_boiler_voltage_ok.Enable := true;
   ZDSV_after_boiler_limit_rotational_moment.Enable := true;
   Burner_flame.N_module := 4;
   Burner_flame.N_chanel := 1;
   Igniter_flame.N_module := 4;
   Igniter_flame.N_chanel := 2;
   KB_close.N_module := 4;
   KB_close.N_chanel := 3;
   KO_open.N_module := 4;
   KO_open.N_chanel := 4;
   KZ_open.N_module := 4;
   KZ_open.N_chanel := 5;
   PZK1_open.N_module := 4;
   PZK1_open.N_chanel := 6;
   PZK2_not_close.N_module := 4;
   PZK2_not_close.N_chanel := 7;
   P_gas_before_BG_min.N_module := 4;
   P_gas_before_BG_min.N_chanel := 8;
   P_gas_before_BG_max.N_module := 4;
   P_gas_before_BG_max.N_chanel := 9;
   P_air_before_burner_min.N_module := 4;
   P_air_before_burner_min.N_chanel := 10;
   P_gas_before_burner_min.N_module := 4;
   P_gas_before_burner_min.N_chanel := 11;
   P_gas_before_burner_max.N_module := 4;
   P_gas_before_burner_max.N_chanel := 12;
   ZRG_open.N_module := 4;
   ZRG_open.N_chanel := 13;
   ZRG_close.N_module := 4;
   ZRG_close.N_chanel := 14;
   ZRG_middle.N_module := 4;
   ZRG_middle.N_chanel := 15;
   ZRG_avto.N_module := 4;
   ZRG_avto.N_chanel := 16;
   NAV_open.N_module := 5;
   NAV_open.N_chanel := 1;
   NAV_close.N_module := 5;
   NAV_close.N_chanel := 2;
   NAV_middle.N_module := 5;
   NAV_middle.N_chanel := 3;
   NAV_avto.N_module := 5;
   NAV_avto.N_chanel := 4;
   NAD_open.N_module := 5;
   NAD_open.N_chanel := 5;
   NAD_close.N_module := 5;
   NAD_close.N_chanel := 6;
   NAD_middle.N_module := 5;
   NAD_middle.N_chanel := 7;
   NAD_avto.N_module := 5;
   NAD_avto.N_chanel := 8;
   dP_furnace_boiler_min.N_module := 5;
   dP_furnace_boiler_min.N_chanel := 9;
   T_water_after_boiler_max.N_module := 5;
   T_water_after_boiler_max.N_chanel := 10;
   Q_water_boiler_min.N_module := 5;
   Q_water_boiler_min.N_chanel := 11;
   Q_water_boiler_max.N_module := 5;
   Q_water_boiler_max.N_chanel := 12;
   P_water_after_boiler_min.N_module := 5;
   P_water_after_boiler_min.N_chanel := 13;
   P_water_after_boiler_max.N_module := 5;
   P_water_after_boiler_max.N_chanel := 14;
   P_water_before_boiler_min.N_module := 5;
   P_water_before_boiler_min.N_chanel := 15;
   P_water_before_boiler_max.N_module := 5;
   P_water_before_boiler_max.N_chanel := 16;
   Call_power_supply_сabinet.N_module := 6;
   Call_power_supply_сabinet.N_chanel := 1;
   DV_Invertor_alarm.N_module := 6;
   DV_Invertor_alarm.N_chanel := 2;
   DV_local_control.N_module := 6;
   DV_local_control.N_chanel := 3;
   DV_dist_control.N_module := 6;
   DV_dist_control.N_chanel := 4;
   DV_powergrid_mode.N_module := 6;
   DV_powergrid_mode.N_chanel := 5;
   DV_invertor_mode.N_module := 6;
   DV_invertor_mode.N_chanel := 6;
   DV_invertor_QF_on.N_module := 6;
   DV_invertor_QF_on.N_chanel := 7;
   DV_powergrid_QF_on.N_module := 6;
   DV_powergrid_QF_on.N_chanel := 8;
   DV_invertor_on.N_module := 6;
   DV_invertor_on.N_chanel := 9;
   DV_powergrid_on.N_module := 6;
   DV_powergrid_on.N_chanel := 10;
   DV_no_voltage.N_module := 6;
   DV_no_voltage.N_chanel := 11;
   DS_Invertor_alarm.N_module := 6;
   DS_Invertor_alarm.N_chanel := 12;
   DS_local_control.N_module := 6;
   DS_local_control.N_chanel := 13;
   DS_dist_control.N_module := 6;
   DS_dist_control.N_chanel := 14;
   DS_powergrid_mode.N_module := 6;
   DS_powergrid_mode.N_chanel := 15;
   DS_invertor_mode.N_module := 6;
   DS_invertor_mode.N_chanel := 16;
   DS_invertor_QF_on.N_module := 7;
   DS_invertor_QF_on.N_chanel := 1;
   DS_powergrid_QF_on.N_module := 7;
   DS_powergrid_QF_on.N_chanel := 2;
   DS_invertor_on.N_module := 7;
   DS_invertor_on.N_chanel := 3;
   DS_powergrid_on.N_module := 7;
   DS_powergrid_on.N_chanel := 4;
   DS_no_voltage.N_module := 7;
   DS_no_voltage.N_chanel := 5;
   CO_1.N_module := 7;
   CO_1.N_chanel := 6;
   CO_2.N_module := 7;
   CO_2.N_chanel := 7;
   CH4.N_module := 7;
   CH4.N_chanel := 8;
   Btn_STOP.Enable := true;
   Btn_STOP.N_module := 7;
   Btn_STOP.N_chanel := 9;
   Btn_Ventilation.Enable := true;
   Btn_Ventilation.N_module := 7;
   Btn_Ventilation.N_chanel := 10;
   Btn_Ignition.Enable := true;
   Btn_Ignition.N_module := 7;
   Btn_Ignition.N_chanel := 11;
   Btn_Sound.Enable := true;
   Btn_Sound.N_module := 7;
   Btn_Sound.N_chanel := 12;
   SHEU_voltage_ok.N_module := 7;
   SHEU_voltage_ok.N_chanel := 13;
   PZK2_open.N_module := 7;
   PZK2_open.N_chanel := 14;
   Power_PLC_from_UPS.N_module := 7;
   Power_PLC_from_UPS.N_chanel := 15;
   UPS_Low_charge.Enable := true;
   UPS_Low_charge.N_module := 7;
   UPS_Low_charge.N_chanel := 16;
   ZRG_voltage_ok.N_module := 8;
   ZRG_voltage_ok.N_chanel := 1;
   NAV_voltage_ok.N_module := 8;
   NAV_voltage_ok.N_chanel := 2;
   NAD_voltage_ok.N_module := 8;
   NAD_voltage_ok.N_chanel := 3;
   ZDG_no_open.N_module := 8;
   ZDG_no_open.N_chanel := 4;
   ZDG_no_close.N_module := 8;
   ZDG_no_close.N_chanel := 5;
   ZDG_opening.N_module := 8;
   ZDG_opening.N_chanel := 6;
   ZDG_closing.N_module := 8;
   ZDG_closing.N_chanel := 7;
   ZDG_voltage_ok.N_module := 8;
   ZDG_voltage_ok.N_chanel := 8;
   ZDSV_before_boiler_no_open.N_module := 8;
   ZDSV_before_boiler_no_open.N_chanel := 9;
   ZDSV_before_boiler_no_close.N_module := 8;
   ZDSV_before_boiler_no_close.N_chanel := 10;
   ZDSV_before_boiler_opening.N_module := 8;
   ZDSV_before_boiler_opening.N_chanel := 11;
   ZDSV_before_boiler_closing.N_module := 8;
   ZDSV_before_boiler_closing.N_chanel := 12;
   ZDSV_before_boiler_voltage_ok.N_module := 8;
   ZDSV_before_boiler_voltage_ok.N_chanel := 13;
   ZDSV_before_boiler_limit_rotational_moment.N_module := 8;
   ZDSV_before_boiler_limit_rotational_moment.N_chanel := 14;
   ZDSV_after_boiler_no_open.N_module := 8;
   ZDSV_after_boiler_no_open.N_chanel := 15;
   ZDSV_after_boiler_no_close.N_module := 8;
   ZDSV_after_boiler_no_close.N_chanel := 16;
   ZDSV_after_boiler_opening.N_module := 9;
   ZDSV_after_boiler_opening.N_chanel := 1;
   ZDSV_after_boiler_closing.N_module := 9;
   ZDSV_after_boiler_closing.N_chanel := 2;
   ZDSV_after_boiler_voltage_ok.N_module := 9;
   ZDSV_after_boiler_voltage_ok.N_chanel := 3;
   ZDSV_after_boiler_limit_rotational_moment.N_module := 9;
   ZDSV_after_boiler_limit_rotational_moment.N_chanel := 4;
   ZRG_control_open.Enable := true;
   ZRG_control_close.Enable := true;
   NAV_control_open.Enable := true;
   NAV_control_close.Enable := true;
   NAD_control_open.Enable := true;
   NAD_control_close.Enable := true;
   Indication_RUN.Enable := true;
   Indication_ALARM.Enable := true;
   Indication_NORMA.Enable := true;
   Indication_READY.Enable := true;
   ZDG_control_open.Enable := true;
   ZDG_control_close.Enable := true;
   ZDG_control_stop.Enable := true;
   ZDG_control_disable_open.Enable := true;
   KB_control_close.Enable := true;
   KO_control_open.Enable := true;
   KZ_control_open.Enable := true;
   IVN_control_on.Enable := true;
   PZK1_control_open.Enable := true;
   PZK2_control_open.Enable := true;
   ZDSV_before_boiler_control_open.Enable := true;
   ZDSV_before_boiler_control_close.Enable := true;
   ZDSV_before_boiler_control_stop.Enable := true;
   ZDSV_before_boiler_control_disable_close.Enable := true;
   ZDSV_after_boiler_control_open.Enable := true;
   ZDSV_after_boiler_control_close.Enable := true;
   ZDSV_after_boiler_control_stop.Enable := true;
   ZDSV_after_boiler_control_disable_close.Enable := true;
   control_alarm_signal.Enable := true;
   DV_control_start.Enable := true;
   DV_control_stop.Enable := true;
   DS_control_start.Enable := true;
   DS_control_stop.Enable := true;
   ZRG_control_open.N_module := 10;
   ZRG_control_open.N_chanel := 1;
   ZRG_control_close.N_module := 10;
   ZRG_control_close.N_chanel := 2;
   NAV_control_open.N_module := 10;
   NAV_control_open.N_chanel := 3;
   NAV_control_close.N_module := 10;
   NAV_control_close.N_chanel := 4;
   NAD_control_open.N_module := 10;
   NAD_control_open.N_chanel := 5;
   NAD_control_close.N_module := 10;
   NAD_control_close.N_chanel := 6;
   Indication_RUN.N_module := 10;
   Indication_RUN.N_chanel := 7;
   Indication_ALARM.N_module := 10;
   Indication_ALARM.N_chanel := 8;
   Indication_NORMA.N_module := 10;
   Indication_NORMA.N_chanel := 9;
   Indication_READY.N_module := 10;
   Indication_READY.N_chanel := 10;
   ZDG_control_open.N_module := 11;
   ZDG_control_open.N_chanel := 1;
   ZDG_control_close.N_module := 11;
   ZDG_control_close.N_chanel := 2;
   ZDG_control_stop.N_module := 11;
   ZDG_control_stop.N_chanel := 3;
   ZDG_control_disable_open.N_module := 11;
   ZDG_control_disable_open.N_chanel := 4;
   KB_control_close.N_module := 11;
   KB_control_close.N_chanel := 5;
   KO_control_open.N_module := 11;
   KO_control_open.N_chanel := 6;
   KZ_control_open.N_module := 11;
   KZ_control_open.N_chanel := 7;
   IVN_control_on.N_module := 11;
   IVN_control_on.N_chanel := 8;
   PZK1_control_open.N_module := 11;
   PZK1_control_open.N_chanel := 9;
   PZK2_control_open.N_module := 11;
   PZK2_control_open.N_chanel := 10;
   ZDSV_before_boiler_control_open.N_module := 11;
   ZDSV_before_boiler_control_open.N_chanel := 11;
   ZDSV_before_boiler_control_close.N_module := 11;
   ZDSV_before_boiler_control_close.N_chanel := 12;
   ZDSV_before_boiler_control_stop.N_module := 11;
   ZDSV_before_boiler_control_stop.N_chanel := 13;
   ZDSV_before_boiler_control_disable_close.N_module := 11;
   ZDSV_before_boiler_control_disable_close.N_chanel := 14;
   ZDSV_after_boiler_control_open.N_module := 11;
   ZDSV_after_boiler_control_open.N_chanel := 15;
   ZDSV_after_boiler_control_close.N_module := 11;
   ZDSV_after_boiler_control_close.N_chanel := 16;
   ZDSV_after_boiler_control_stop.N_module := 12;
   ZDSV_after_boiler_control_stop.N_chanel := 1;
   ZDSV_after_boiler_control_disable_close.N_module := 12;
   ZDSV_after_boiler_control_disable_close.N_chanel := 2;
   control_alarm_signal.N_module := 12;
   control_alarm_signal.N_chanel := 3;
   DV_control_start.N_module := 12;
   DV_control_start.N_chanel := 4;
   DV_control_stop.N_module := 12;
   DV_control_stop.N_chanel := 5;
   DS_control_start.N_module := 12;
   DS_control_start.N_chanel := 6;
   DS_control_stop.N_module := 12;
   DS_control_stop.N_chanel := 7;
   DV_control_frequency.Enable := true;
   DS_control_frequency.Enable := true;
   DV_control_frequency.N_module := 13;
   DV_control_frequency.N_chanel := 1;
   DS_control_frequency.N_module := 13;
   DS_control_frequency.N_chanel := 2;
   T_gas_before_BG.Enable := false;
   P_gas_before_BG.Enable := false;
   Btn_STOP.Invert := true;
   DV_no_voltage.Invert := true;
   DS_no_voltage.Invert := true;
   DS_control_frequency.High_limit_phisical_new := 50.0;
   DS_control_frequency.High_limit_phisical_current := 50.0;
   DV_control_frequency.High_limit_phisical_current := 50.0;
   DV_control_frequency.High_limit_phisical_new := 50.0;
   NAV_position.Low_limit_ADC_current := 577;
   NAV_position.High_limit_ADC_current := 17374;
   NAV_position.Low_limit_ADC_new := 577;
   NAV_position.High_limit_ADC_new := 17374;
   NAD_position.Low_limit_ADC_current := 1732;
   NAD_position.High_limit_ADC_current := 25516;
   NAD_position.Low_limit_ADC_new := 1732;
   NAD_position.High_limit_ADC_new := 25516;
   ZRG_position.Low_limit_ADC_current := 4531;
   ZRG_position.Low_limit_ADC_new := 4531;
   ZRG_position.High_limit_ADC_current := 17131;
   ZRG_position.High_limit_ADC_new := 17131;
   Q_water_boiler.Enable := true;
   Q_gas.Enable := true;
   Q_gas.Tgas_fixed_value_on := true;
   Q_gas.Tgas_fixed_value := -4.0;
   Q_gas.Pgas_fixed_value_on := true;
   Q_gas.Pgas_fixed_value := 141.3232;
END_DATA_BLOCK

DATA_BLOCK "Alarms_and_warnings"   // DB2
{ S7_Optimized_Access := 'FALSE' }
VERSION : 0.1
   VAR
      Reset_alarms : Bool;   // Сброс аварий и предупреждений
      Warning_sensor_T_water_before_boiler : Bool;   // Предупреждение. Неисправность датчика T сетевой воды перед котлом
      Warning_sensor_P_water_before_boiler : Bool;   // Предупреждение. Неисправность датчика P сетевой воды перед котлом
      Warning_sensor_dP_water_boiler : Bool;   // Предупреждение. Неисправность датчика dP сетевой воды через котел
      Warning_sensor_T_water_after_boiler : Bool;   // Предупреждение. Неисправность датчика Т сетевой воды после котла
      Warning_sensor_P_water_after_boiler : Bool;   // Предупреждение. Неисправность датчика P сетевой воды после котла
      Warning_sensor_dP_water_boiler_1 : Bool;   // Предупреждение. Неисправность датчика dP сетевой воды через котел
      Warning_sensor_P_water_before_boiler_1 : Bool;   // Предупреждение. Неисправность датчика P сетевой воды перед котлом
      Warning_sensor_dP_gas_boiler : Bool;   // Предупреждение. Неисправность датчика dP газа на котел
      Warning_sensor_dP_furnace_boiler : Bool;   // Предупреждение. Неисправность датчика разрежения в топке котла
      Warning_sensor_P_gas_before_PZK1_and_PZK2 : Bool;   // Предупреждение. Неисправность датчика P газа между ПЗК-1 и ПЗК-2
      Warning_sensor_P_gas_before_burner : Bool;   // Предупреждение. Неисправность датчика P газа перед горелкой
      Warning_sensor_P_air_burner : Bool;   // Предупреждение. Неисправность датчика P воздуха к горелке
      Warning_sensor_T_exhaust_gas : Bool;   // Предупреждение. Неисправность датчика T уходящих газов
      Warning_sensor_ZRG_position : Bool;   // Предупреждение. Неисправность датчика положения рег. заслонки газа перед котлом
      Warning_sensor_NAV_position : Bool;   // Предупреждение. Неисправность датчика положения направл. аппарата вентилятора
      Warning_sensor_NAD_position : Bool;   // Предупреждение. Неисправность датчика положения направл. аппарата дымососа
      Warning_sensor_DV_current_frequency : Bool;   // Предупреждение. Неисправность датчика Текущ. значение ПЧ ДВ
      Warning_sensor_DS_current_frequency : Bool;   // Предупреждение. Неисправность датчика Текущ. значение ПЧ ДС
      Warning_ZDSV_before_boiler_limit_rotational_moment : Bool;   // Предупреждение. Сработал ограничитель крутящего момента ЗДСВ перед котлом
      Warning_ZDSV_after_boiler_limit_rotational_moment : Bool;   // Предупреждение. Сработал ограничитель крутящего момента ЗДСВ после котла
      Warning_сall_power_supply_сabinet : Bool;   // Предупреждение. Вызов к шкафу электропитания
      Warning_DV_need_on_QF_invertor : Bool;   // Предупреждение. ДВ. Необходимо включить QF ПЧ
      Warning_DV_need_on_QF_powergrid : Bool;   // Предупреждение. ДВ. Необходимо включить QF Сети
      Warning_DV_no_voltage : Bool;   // Предупреждение. ДВ. Неисправность напряжения в сети ШУД
      Warning_DS_need_on_QF_invertor : Bool;   // Предупреждение. ДС. Необходимо включить QF ПЧ
      Warning_DS_need_on_QF_powergrid : Bool;   // Предупреждение. ДС. Необходимо включить QF Сети
      Warning_DS_no_voltage : Bool;   // Предупреждение. ДС. Неисправность напряжения в сети ШУД
      Warning_SHEU_no_voltage : Bool;   // Предупреждение. Нет питания ШЭУ
      Warning_power_PLC_from_UPS : Bool;   // Предупреждение. Питание контроллера от ИБП
      Warning_UPS_Low_charge : Bool;   // Предупреждение. Низкий заряд батареи ИБП
      Warning_ZRG_no_voltage : Bool;   // Предупреждение. Нет питания ЗРГ
      Warning_ZDG_no_voltage : Bool;   // Предупреждение. Нет питания ЗДГ
      Warning_NAV_no_voltage : Bool;   // Предупреждение. Нет питания НАВ
      Warning_NAD_no_voltage : Bool;   // Предупреждение. Нет питания НАД
      Warning_ZDSV_before_boiler_no_voltage : Bool;   // Предупреждение. Нет питания ЗДСВ перед котлом
      Warning_ZDSV_after_boiler_no_voltage : Bool;   // Предупреждение. Нет питания ЗДСВ после котла
      Warning_DV_invertor_alarm : Bool;   // Предупреждение. Авария ПЧ ДВ
      Warning_DS_invertor_alarm : Bool;   // Предупреждение. Авария ПЧ ДС
      Warning_ZRG_manual : Bool;   // Предупреждение. ЗРГ в местном режиме
      Warning_NAV_manual : Bool;   // Предупреждение. НАВ в местном режиме
      Warning_NAD_manual : Bool;   // Предупреждение. НАД в местном режиме
      Warning_DV_manual : Bool;   // Предупреждение. ДВ в местном режиме
      Warning_DS_manual : Bool;   // Предупреждение. ДС в местном режиме
      Alarm_P_gas_before_BG_max : Bool;   // Повышение давления газа перед БГ
      Enable_Alarm_P_gas_before_BG_max : Bool;   // Разрешение аварии. Повышение давления газа перед БГ
      TIME_Alarm_P_gas_before_BG_max : Int := 5;   // Время формирования аварии. Повышение давления газа перед БГ (сек)
      Alarm_P_gas_before_BG_min : Bool;   // Понижение давления газа перед БГ
      Enable_Alarm_P_gas_before_BG_min : Bool;   // Разрешение аварии. Понижение давления газа перед БГ
      TIME_Alarm_P_gas_before_BG_min : Int := 5;   // Время формирования аварии. Понижение давления газа перед БГ (сек)
      Alarm_P_gas_before_burner_min : Bool;   // Понижение давления газа перед горелкой
      Enable_Alarm_P_gas_before_burner_min : Bool;   // Разрешение аварии. Понижение давления газа перед горелкой
      TIME_Alarm_P_gas_before_burner_min : Int := 5;   // Время формирования аварии. Понижение давления газа перед горелкой (сек)
      Alarm_P_gas_before_burner_max : Bool;   // Повышение давления газа перед горелкой
      Enable_Alarm_P_gas_before_burner_max : Bool;   // Разрешение аварии. Повышение давления газа перед горелкой
      TIME_Alarm_P_gas_before_burner_max : Int := 5;   // Время формирования аварии. Повышение давления газа перед горелкой (сек)
      Alarm_DS_off : Bool;   // Отключение ДС
      Enable_Alarm_DS_off : Bool;   // Разрешение аварии. Отключение ДС
      TIME_Alarm_DS_off : Int := 1;   // Время формирования аварии. Отключение ДС (сек)
      Alarm_DV_off : Bool;   // Отключение ДВ
      Enable_Alarm_DV_off : Bool;   // Разрешение аварии. Отключение ДВ
      TIME_Alarm_DV_off : Int := 1;   // Время формирования аварии. Отключение ДВ (сек)
      Alarm_dP_furnace_boiler_min : Bool;   // Понижение разряжения в топке
      Enable_Alarm_dP_furnace_boiler_min : Bool;   // Разрешение аварии. Понижение разряжения в топке
      TIME_Alarm_dP_furnace_boiler_min : Int := 5;   // Время формирования аварии. Понижение разряжения в топке (сек)
      Alarm_P_air_before_burner_min : Bool;   // Понижение давления воздуха перед горелкой
      Enable_Alarm_P_air_before_burner_min : Bool;   // Разрешение аварии. Понижение давления воздуха перед горелкой
      TIME_Alarm_P_air_before_burner_min : Int := 5;   // Время формирования аварии. Понижение давления воздуха перед горелкой (сек)
      Alarm_P_water_after_boiler_min : Bool;   // Понижение давления сетевой воды за котлом
      Enable_Alarm_P_water_after_boiler_min : Bool;   // Разрешение аварии. Понижение давления сетевой воды за котлом
      TIME_Alarm_P_water_after_boiler_min : Int := 5;   // Время формирования аварии. Понижение давления сетевой воды за котлом (сек)
      Alarm_P_water_after_boiler_max : Bool;   // Повышение давления сетевой воды за котлом
      Enable_Alarm_P_water_after_boiler_max : Bool;   // Разрешение аварии. Повышение давления сетевой воды за котлом
      TIME_Alarm_P_water_after_boiler_max : Int := 5;   // Время формирования аварии. Повышение давления сетевой воды за котлом (сек)
      Alarm_T_water_after_boiler_max : Bool;   // Повышение температуры сетевой воды за котлом
      Enable_Alarm_T_water_after_boiler_max : Bool;   // Разрешение аварии. Повышение температуры сетевой воды за котлом
      TIME_Alarm_T_water_after_boiler_max : Int := 5;   // Время формирования аварии. Повышение температуры сетевой воды за котлом (сек)
      Alarm_Q_water_boiler_min : Bool;   // Понижение расхода сетевой воды через котел
      Enable_Alarm_Q_water_boiler_min : Bool;   // Разрешение аварии. Понижение расхода сетевой воды через котел
      TIME_Alarm_Q_water_boiler_min : Int := 5;   // Время формирования аварии. Понижение расхода сетевой воды через котел (сек)
      Alarm_Not_flame_burner : Bool := false;   // Невоспламенение или погасание факела горелки котла
      Enable_Alarm_Not_flame_burner : Bool := false;   // Разрешение аварии. Невоспламенение или погасание факела горелки котла
      TIME_Alarm_Not_flame_burner : Int := 50;   // Время формирования аварии. Невоспламенение или погасание факела горелки котла (мсек)
      Alarm_stop_HMI : Bool := false;   // Нажата кнопка аварийного останова на панели оператора
      Enable_Alarm_stop_HMI : Bool := false;   // Разрешение аварии. Нажата кнопка аварийного останова на панели оператора
      Alarm_stop_SCADA : Bool := false;   // Нажата кнопка аварийного останова на SCADA
      Enable_Alarm_stop_SCADA : Bool := false;   // Разрешение аварии. Нажата кнопка аварийного останова на SCADA
      Alarm_CO2_porog2 : Bool := false;   // СО2 порог 2
      Enable_Alarm_CO2_porog2 : Bool := true;   // Разрешение аварии. СО2 порог 2
      TIME_Alarm_CO2_porog2 : Int := 5;   // Время формирования аварии. СО2 порог 2 (сек)
      Alarm_CH4 : Bool := false;   // CH4
      Enable_Alarm_CH4 : Bool := true;   // Разрешение аварии. CH4
      TIME_Alarm_CH4 : Int := 5;   // Время формирования аварии. CH4 (сек)
      Warning_Not_flame_Igniter : Bool := false;   // Предупреждение. Пламя запальника потухло
      Enable_Warning_Not_flame_Igniter : Bool := false;   // Разрешение предупреждения. Пламя запальника потухло
      TIME_Warning_Not_flame_Igniter : Int := 300;   // Время формирования предупреждения. Пламя запальника потухло (мсек)
      Warning_PZK2_not_open : Bool := false;   // Предупреждение. ПЗК2 не открылся
      Enable_Warning_PZK2_not_open : Bool := false;   // Разрешение предупреждения. ПЗК2 не открылся
      TIME_Warning_PZK2_not_open : Int := 55;   // Время формирования предупреждения. ПЗК2 не открылся (сек)
      Global_alarm : Bool;   // Обобщенный признак аварии
      SP_alarm_H_P_gas_before_BG : Real := 37.0;   // Аварийная уставка. Высокое давление газа перед БГ
      SP_alarm_L_P_gas_before_BG : Real := 5.0;   // Аварийная уставка. Низкое давление газа перед БГ
      SP_warning_H_P_gas_before_BG : Real;   // Предупредительная уставка. Высокое давление газа перед БГ
      SP_warning_L_P_gas_before_BG : Real;   // Предупредительная уставка. Низкое давление газа перед БГ
      SP_alarm_H_P_gas_before_burner : Real := 30.5;   // Аварийная уставка. Высокое давление газа перед горелкой
      SP_alarm_L_P_gas_before_burner : Real := 0.04;   // Аварийная уставка. Низкое давление газа перед горелкой
      SP_warning_H_P_gas_before_burner : Real;   // Предупредительная уставка. Высокое давление газа перед горелкой
      SP_warning_L_P_gas_before_burner : Real;   // Предупредительная уставка. Низкое давление газа перед горелкой
      SP_alarm_H_P_air_before_burner : Real;   // Аварийная уставка. Высокое давление воздуха перед горелкой
      SP_alarm_L_P_air_before_burner : Real := 15.0;   // Аварийная уставка. Низкое давление воздуха перед горелкой
      SP_warning_H_P_air_before_burner : Real;   // Предупредительная уставка. Высокое давление воздуха перед горелкой
      SP_warning_L_P_air_before_burner : Real;   // Предупредительная уставка. Низкое давление воздуха перед горелкой
      SP_alarm_H_dP_furnace_boiler : Real;   // Аварийная уставка. Высокое разрежение в топке
      SP_alarm_L_dP_furnace_boiler : Real;   // Аварийная уставка. Низкое разрежение в топке
      SP_warning_H_dP_furnace_boiler : Real;   // Предупредительная уставка. Высокое разрежение в топке
      SP_warning_L_dP_furnace_boiler : Real;   // Предупредительная уставка. Низкое разрежение в топке
      SP_alarm_H_P_water_before_boiler : Real;   // Аварийная уставка. Высокое давление воды перед котлом
      SP_alarm_L_P_water_before_boiler : Real;   // Аварийная уставка. Низкое давление воды перед котлом
      SP_warning_H_P_water_before_boiler : Real := 11.5;   // Предупредительная уставка. Высокое давление воды перед котлом
      SP_warning_L_P_water_before_boiler : Real := 4.5;   // Предупредительная уставка. Низкое давление воды перед котлом
      SP_alarm_H_P_water_after_boiler : Real := 12.2;   // Аварийная уставка. Высокое давление воды после котла
      SP_alarm_L_P_water_after_boiler : Real := 3.3;   // Аварийная уставка. Низкое давление воды после котла
      SP_warning_H_P_water_after_boiler : Real := 11.5;   // Предупредительная уставка. Высокое давление воды после котла
      SP_warning_L_P_water_after_boiler : Real := 3.9;   // Предупредительная уставка. Низкое давление воды после котла
      SP_alarm_H_T_water_after_boiler : Real := 125.0;   // Аварийная уставка. Высокая температура воды после котла
      SP_alarm_L_T_water_after_boiler : Real;   // Аварийная уставка. Низкая температура воды после котла
      SP_warning_H_T_water_after_boiler : Real := 115.0;   // Предупредительная уставка. Высокая температура воды после котла
      SP_warning_L_T_water_after_boiler : Real;   // Предупредительная уставка. Низкая температура воды после котла
      SP_alarm_H_Q_water_boiler : Real;   // Аварийная уставка. Высокий расход сетевой воды через котел
      SP_alarm_L_Q_water_boiler : Real := 100.0;   // Аварийная уставка. Низкий расход сетевой воды через котел
      SP_warning_H_Q_water_boiler : Real := 240.0;   // Предупредительная уставка. Высокий расход сетевой воды через котел
      SP_warning_L_Q_water_boiler : Real := 130.0;   // Предупредительная уставка. Низкий расход сетевой воды через котел
      Warning_P_water_before_boiler_min : Bool;   // Понижение давления сетевой воды перед котлом
      Warning_P_water_before_boiler_max : Bool;   // Повышение давления сетевой воды перед котлом
      Warning_P_water_after_boiler_min : Bool;   // Понижение давления сетевой воды после котла
      Warning_P_water_after_boiler_max : Bool;   // Повышение давления сетевой воды после котла
      Warning_T_water_after_boiler_max : Bool;   // Повышение температуры сетевой воды после котла
      Warning_Q_water_boiler_max : Bool;   // Повышение расхода сетевой воды через котел
      Warning_Q_water_boiler_min : Bool;   // Понижение расхода сетевой воды через котел
      Warning_CO2_porog1 : Bool := false;   // СО2 порог 1
      Warning_sensor_P_gas_before_BG : Bool;   // Предупреждение. Неисправность датчика P газа перед БГ
      Warning_dP_furnace_boiler_min : Bool;   // Предупреждение. Понижение разряжения в топке
      Warning_P_air_before_burner_min : Bool;   // Предупреждение. Понижение давления воздуха перед горелкой
      Warning_ZDG_not_close : Bool := false;   // Предупреждение. ЗДГ не закрылся
      Enable_Warning_ZDG_not_close : Bool := false;   // Разрешение предупреждения. ЗДГ не закрылся
      TIME_Warning_ZDG_not_close : Int := 30;   // Время формирования предупреждения. ЗДГ не закрылся (сек)
      Warning_protection_block : Bool;   // Предупреждение. Имеется блокировка защиты
   END_VAR
BEGIN
END_DATA_BLOCK

DATA_BLOCK "Protections"   // DB3
{ S7_Optimized_Access := 'FALSE' }
VERSION : 0.1
   VAR
      Global : Bool;   // Сработка защиты
      P_gas_before_BG_max : Bool;   // Повышение давления газа перед БГ
      P_gas_before_BG_min : Bool;   // Понижение давления газа перед БГ
      P_gas_before_burner_min : Bool;   // Понижение давления газа перед горелкой
      P_gas_before_burner_max : Bool;   // Повышение давления газа перед горелкой
      DS_off : Bool;   // Отключение ДС
      DV_off : Bool;   // Отключение ДВ
      dP_in_furnance_min : Bool;   // Понижение разряжения в топке
      P_air_before_burner_min : Bool;   // Понижение давления воздуха перед горелкой
      P_water_after_boiler_min : Bool;   // Понижение давления сетевой воды за котлом
      P_water_after_boiler_max : Bool;   // Повышение давления сетевой воды за котлом
      T_water_after_boiler_max : Bool;   // Повышение температуры сетевой воды за котлом
      Q_water_boiler_min : Bool;   // Понижение расхода сетевой воды через котел
      Not_flame_burner : Bool;   // Невоспламенение или погасание факела горелки котла
      Alarm_stop_HMI : Bool;   // Нажата кнопка аварийного останова на панели операторора
      Alarm_stop_SCADA : Bool;   // Нажата кнопка аварийного останова на SCADA
      CO2_porog2 : Bool;   // СО2 порог 2
      CH4 : Bool;   // CH4
      BLOCK_P_gas_before_BG_max : Bool;   // БЛОКИРОВКА. Повышение давления газа перед БГ
      BLOCK_P_gas_before_BG_min : Bool;   // БЛОКИРОВКА. Понижение давления газа перед БГ
      BLOCK_P_gas_before_burner_min : Bool;   // БЛОКИРОВКА. Понижение давления газа перед горелкой
      BLOCK_P_gas_before_burner_max : Bool;   // БЛОКИРОВКА. Повышение давления газа перед горелкой
      BLOCK_DS_off : Bool;   // БЛОКИРОВКА. Отключение ДС
      BLOCK_DV_off : Bool;   // БЛОКИРОВКА. Отключение ДВ
      BLOCK_dP_in_furnance_min : Bool;   // БЛОКИРОВКА. Понижение разряжения в топке
      BLOCK_P_air_before_burner_min : Bool;   // БЛОКИРОВКА. Понижение давления воздуха перед горелкой
      BLOCK_P_water_after_boiler_min : Bool;   // БЛОКИРОВКА. Понижение давления сетевой воды за котлом
      BLOCK_P_water_after_boiler_max : Bool;   // БЛОКИРОВКА. Повышение давления сетевой воды за котлом
      BLOCK_T_water_after_boiler_max : Bool;   // БЛОКИРОВКА. Повышение температуры сетевой воды за котлом
      BLOCK_Q_water_boiler_min : Bool;   // БЛОКИРОВКА. Понижение расхода сетевой воды через котел
      BLOCK_Not_flame_burner : Bool;   // БЛОКИРОВКА. Невоспламенение или погасание факела горелки котла
      BLOCK_Alarm_stop_HMI : Bool;   // БЛОКИРОВКА. Нажата кнопка аварийного останова на панели операторора
      BLOCK_Alarm_stop_SCADA : Bool;   // БЛОКИРОВКА. Нажата кнопка аварийного останова на SCADA
      BLOCK_CO2_porog2 : Bool;   // БЛОКИРОВКА. СО2 порог 2
      BLOCK_CH4 : Bool;   // БЛОКИРОВКА. CH4
   END_VAR
BEGIN
END_DATA_BLOCK

DATA_BLOCK "Technology"   // DB4
{ S7_Optimized_Access := 'FALSE' }
VERSION : 0.1
   VAR
      Regim : USInt;   // Текущий режим работы
      Regim_off_step : USInt;   // Режим ОТКЛ. Текущий шаг
      Regim_check_step : USInt;   // Режим ПРОВЕРКА. Текущий шаг
      Regim_ventilation_step : USInt;   // Режим ВЕНТИЛЯЦИЯ. Текущий шаг
      Regim_press_step : USInt;   // Режим ОПРЕССОВКА. Текущий шаг
      Regim_ignition_step : USInt;   // Режим РОЗЖИГ. Текущий шаг
      Regim_min_power_step : USInt;   // Режим ВЫХОД НА МИН МОЩНОСТЬ. Текущий шаг
      Regim_heating_step : USInt;   // Режим ПРОГРЕВ. Текущий шаг
      Regim_run_step : USInt;   // Режим РАБОТА. Текущий шаг
      Regim_emergency_stop_step : USInt;   // Режим ЭКСТРЕННЫЙ ОСТАНОВ. Текущий шаг
      Regim_alarm_stop_step : USInt;   // Режим АВАРИЙНЫЙ ОСТАНОВ. Текущий шаг
      Regim_plan_stop_step : USInt;   // Режим ПЛАНОВЫЙ ОСТАНОВ. Текущий шаг
      Regim_stop_press_step : USInt;   // Режим ПОСТОСТАНОВОЧНАЯ ОПРЕССОВКА. Текущий шаг
      Regim_short_ventilation_step : USInt;   // Режим УКОРОЧЕННАЯ ВЕНТИЛЯЦИЯ. Текущий шаг
      Regim_test_press_step : USInt;   // Режим ТЕСТОВАЯ ОПРЕССОВКА. Текущий шаг
      Regim_test_ignition_step : USInt;   // Режим ТЕСТОВЫЙ РОЗЖИГ. Текущий шаг
      SP_TIME_Ventilation : Int := 600;   // Уставка времени вентиляции топки перед розжигом (сек)
      SP_TIME_Ventilation_start : Int := 5;   // Уставка времени определения начала вентиляции (сек)
      DB_P_air_ventilation : Int := 15;   // Допустимое отклонение P воздуха при вентиляции (%)
      DB_dP_furnace_ventilation : Int := 15;   // Допустимое отклонение разрежения в топке при вентиляции (%)
      DB_P_air_ignition : Int := 20;   // Допустимое отклонение P воздуха при розжиге (%)
      DB_dP_furnace_ignition : Int := 20;   // Допустимое отклонение разряжения в топке при розжиге (%)
      SP_TIME_check_P_between_PZK : Int := 5;   // Уставка времени проверки давления между ПЗК при опрессовке (сек)
      SP_P_between_PZK_check_max : Real := 15.0;   // Уставка MAX Давления между ПЗК при опрессовке
      SP_P_between_PZK_check_min : Real := 6.0;   // Уставка MIN Давления между ПЗК при опрессовке
      CNT_Igniter : Int;   // Счетчик попыток розжига запальника
      Heating_enable : Bool := true;   // Разрешение режима ПРОГРЕВ
      Max_P_gas_heating : Real := 1.2;   // Max давления газа для режима прогрев
      SP_TIME_Heating : Int := 3;   // Уставка времени прогрева (мин)
      SP_T_water_after_boiler : Real := 72.0;   // Уставка Т воды после котла
      Stop_press_enable : Bool := true;   // Разрешение режима ПОСТОСТАНОВОЧНАЯ ОПРЕССОВКА
      SP_TIME_check_P_stop_press_min : Int := 5;   // Уставка времени проверки давления между ПЗК на min при постостановочной опрессовке (сек)
      SP_TIME_check_P_stop_press_max : Int := 5;   // Уставка времени проверки давления между ПЗК на max при постостановочной опрессовке (сек)
      SP_TIME_Short_ventilation : Int := 120;   // Уставка времени укороченной вентиляции топки (сек)
      Ventilation_conducted : Bool;   // Вентиляция проведена
      Test_press_run : Bool;   // Запущена тестовая опрессовка
      Short_ventilation_enable : Bool := true;   // Разрешение проведения УКОРОЧЕННОЙ ВЕНТИЛЯЦИИ
      Test_ignition_run : Bool;   // Запущен тестовый розжиг
      Substage : Int;   // Подрежим
      transition_ignition : Bool;   // Был переход в розжиг и откытие ПЗК2
      need_plan_stop : Bool;   // Необходимость планового останова
   END_VAR
BEGIN
END_DATA_BLOCK

DATA_BLOCK "HMI"   // DB20
{ S7_Optimized_Access := 'FALSE' }
VERSION : 0.1
   VAR
      Btn_Ventilation_HMI : Bool;   // Кнопка ВЕНТИЛЯЦИЯ на панели оператора
      Btn_Ventilation_SCADA : Bool;   // Кнопка ВЕНТИЛЯЦИЯ на SCADA
      Btn_Ignition_HMI : Bool;   // Кнопка РОЗЖИГ на панели оператора
      Btn_Ignition_SCADA : Bool;   // Кнопка РОЗЖИГ на SCADA
      Btn_normal_stop_HMI : Bool;   // Кнопка НОРМАЛЬНЫЙ ОСТАНОВ на панели оператора
      Btn_normal_stop_SCADA : Bool;   // Кнопка НОРМАЛЬНЫЙ ОСТАНОВ на SCADA
      Btn_alarm_stop_HMI : Bool;   // Кнопка АВАРИЙНЫЙ ОСТАНОВ на панели оператора
      Btn_alarm_stop_SCADA : Bool;   // Кнопка АВАРИЙНЫЙ ОСТАНОВ на SCADA
      Current_SP_P_air : Real;   // Текущая уставка регулятора давления воздуха
      Current_SP_dP_furnance : Real;   // Текущая уставка регулятора разрежения
      Btn_test_press_HMI : Bool;   // Кнопка ТЕСТОВАЯ ОПРЕССОВКА на панели оператора
      Btn_test_ignition_HMI : Bool;   // Кнопка ТЕСТОВЫЙ РОЗЖИГ на панели оператора
      Btn_manual_ignition_HMI : Bool;   // Кнопка Ручной РОЗЖИГ на панели оператора
      Btn_reset_sound_HMI : Bool;   // Кнопка СБРОС ЗВУКА на панели оператора
      TIME_converter_minute : Int;
      TIME_converter_second : Int;
      LTIME_converter_day : DInt;
      LTIME_converter_hour : Int;
      INDICATION_TIME_1 : USInt;
      INDICATION_TIME_2 : USInt;
      TIME_converter_IN : Time;
      LTIME_converter_IN : LTime;
      Btn_Ventilation_HMI_Log : Bool;   // Кнопка ВЕНТИЛЯЦИЯ на панели оператора для журнала событий
      Btn_Ventilation_SCADA_Log : Bool;   // Кнопка ВЕНТИЛЯЦИЯ на SCADA для журнала событий
      Btn_Ventilation_ShAU_Log : Bool;   // Кнопка ВЕНТИЛЯЦИЯ на ШАУ для журнала событий
      Btn_Ignition_HMI_Log : Bool;   // Кнопка РОЗЖИГ на панели оператора для журнала событий
      Btn_Ignition_SCADA_Log : Bool;   // Кнопка РОЗЖИГ на SCADA для журнала событий
      Btn_Ignition_ShAU_Log : Bool;   // Кнопка РОЗЖИГ на ШАУ для журнала событий
      Btn_normal_stop_HMI_Log : Bool;   // Кнопка НОРМАЛЬНЫЙ ОСТАНОВ на панели оператора для журнала событий
      Btn_normal_stop_SCADA_Log : Bool;   // Кнопка НОРМАЛЬНЫЙ ОСТАНОВ на SCADA для журнала событий
      Btn_alarm_stop_HMI_Log : Bool;   // Кнопка АВАРИЙНЫЙ ОСТАНОВ на панели оператора для журнала событий
      Btn_alarm_stop_SCADA_Log : Bool;   // Кнопка АВАРИЙНЫЙ ОСТАНОВ на SCADA для журнала событий
      Btn_emergency_stop_ShAU_Log : Bool;   // Кнопка ЭКСТРЕННЫЙ ОСТАНОВ на ШАУ для журнала событий
      Btn_test_press_HMI_Log : Bool;   // Кнопка ТЕСТОВАЯ ОПРЕССОВКА на панели оператора для журнала событий
      Btn_test_ignition_HMI_Log : Bool;   // Кнопка ТЕСТОВЫЙ РОЗЖИГ на панели оператора для журнала событий
      Btn_manual_ignition_HMI_Log : Bool;   // Кнопка Ручной РОЗЖИГ на панели оператора для журнала событий
      Btn_reset_sound_HMI_Log : Bool;   // Кнопка СБРОС ЗВУКА на панели оператора для журнала событий
      Reset_alarms_Log : Bool;   // Сброс аварий для журнала событий
      Btn_reset_alarms_ShAU_Log : Bool;   // Сброс аварий на ШАУ для журнала событий
      RegMap_Apply_Log : Bool;   // Режимная карта. Применить. Для журнала событий
      DS_Manual_Start_Log : Bool;   // ДС. Ручное управление. Пуск. Для журнала событий
      DS_Manual_Stop_Log : Bool;   // ДС. Ручное управление. Стоп. Для журнала событий
      DV_Manual_Start_Log : Bool;   // ДВ. Ручное управление. Пуск. Для журнала событий
      DV_Manual_Stop_Log : Bool;   // ДВ. Ручное управление. Стоп. Для журнала событий
      ZDG_Manual_open_Log : Bool;   // ЗДГ. Ручное управление. Открыть. Для журнала событий
      ZDG_Manual_close_Log : Bool;   // ЗДГ. Ручное управление. Закрыть. Для журнала событий
      ZDG_Manual_stop_Log : Bool;   // ЗДГ. Ручное управление. Стоп. Для журнала событий
      ZDSV_after_boiler_Manual_open_Log : Bool;   // ЗДСВ после котла. Ручное управление. Открыть. Для журнала событий
      ZDSV_after_boiler_Manual_close_Log : Bool;   // ЗДСВ после котла. Ручное управление. Закрыть. Для журнала событий
      ZDSV_after_boiler_Manual_stop_Log : Bool;   // ЗДСВ после котла. Ручное управление. Стоп. Для журнала событий
      ZDSV_before_boiler_Manual_open_Log : Bool;   // ЗДСВ перед котлом. Ручное управление. Открыть. Для журнала событий
      ZDSV_before_boiler_Manual_close_Log : Bool;   // ЗДСВ перед котлом. Ручное управление. Закрыть. Для журнала событий
      ZDSV_before_boiler_Manual_stop_Log : Bool;   // ЗДСВ перед котлом. Ручное управление. Стоп. Для журнала событий
   END_VAR
BEGIN
END_DATA_BLOCK

DATA_BLOCK "RT_INFO_DB"   // DB25
{ S7_Optimized_Access := 'FALSE' }
VERSION : 0.1
   VAR
      INFO : LTime;
      Ret_val : Int;
      Cycle : UDInt;   // Текущее время цикла (мс)
      temp : UDInt;
   END_VAR
BEGIN
END_DATA_BLOCK

DATA_BLOCK "PID_impulse_ZRG_DB"   // DB26
{ S7_Optimized_Access := 'FALSE' }
VERSION : 0.1
// stored: InstanceOfName PID_impulse
"PID_impulse"
BEGIN
END_DATA_BLOCK

DATA_BLOCK "PID_impulse_NAV_DB"   // DB27
{ S7_Optimized_Access := 'FALSE' }
VERSION : 0.1
// stored: InstanceOfName PID_impulse
"PID_impulse"
BEGIN
END_DATA_BLOCK

DATA_BLOCK "PID_impulse_NAD_DB"   // DB28
{ S7_Optimized_Access := 'FALSE' }
VERSION : 0.1
// stored: InstanceOfName PID_impulse
"PID_impulse"
BEGIN
END_DATA_BLOCK

DATA_BLOCK "PID_analog_DV_DB"   // DB29
{ S7_Optimized_Access := 'FALSE' }
VERSION : 0.1
// stored: InstanceOfName PID_analog
"PID_analog"
BEGIN
END_DATA_BLOCK

DATA_BLOCK "PID_analog_DS_DB"   // DB30
{ S7_Optimized_Access := 'FALSE' }
VERSION : 0.1
// stored: InstanceOfName PID_analog
"PID_analog"
BEGIN
END_DATA_BLOCK

DATA_BLOCK "RegMap"   // DB39
{ S7_Optimized_Access := 'FALSE' }
VERSION : 0.1
   VAR
      P_gaz_1 : Real := 0.6;   // P газа 1 точка
      P_gaz_2 : Real := 1.0;   // P газа 2 точка
      P_gaz_3 : Real := 2.0;   // P газа 3 точка
      P_gaz_4 : Real := 4.0;   // P газа 4 точка
      P_gaz_5 : Real := 5.0;   // P газа 5 точка
      P_gaz_6 : Real := 7.0;   // P газа 6 точка
      P_gaz_7 : Real := 9.0;   // P газа 7 точка
      P_gaz_8 : Real := 10.0;   // P газа 8 точка
      P_air_ventilation : Real := 80.0;   // Р воздуха Вентиляция
      P_air_ignition : Real := 40.0;   // Р воздуха Розжиг
      P_air_1 : Real := 35.0;   // Р воздуха 1 точка
      P_air_2 : Real := 60.0;   // Р воздуха 2 точка
      P_air_3 : Real := 70.0;   // Р воздуха 3 точка
      P_air_4 : Real := 110.0;   // Р воздуха 4 точка
      P_air_5 : Real := 130.0;   // Р воздуха 5 точка
      P_air_6 : Real := 180.0;   // Р воздуха 6 точка
      P_air_7 : Real := 240.0;   // Р воздуха 7 точка
      P_air_8 : Real := 265.0;   // Р воздуха 8 точка
      dP_furnace_ventilation : Real := -30.0;   // dP в топке Вентиляция
      dP_furnace_ignition : Real := -30.0;   // dP в топке Розжиг
      dP_furnace_1 : Real := -30.0;   // dP в топке 1 точка
      dP_furnace_2 : Real := -30.0;   // dP в топке 2 точка
      dP_furnace_3 : Real := -30.0;   // dP в топке 3 точка
      dP_furnace_4 : Real := -30.0;   // dP в топке 4 точка
      dP_furnace_5 : Real := -30.0;   // dP в топке 5 точка
      dP_furnace_6 : Real := -30.0;   // dP в топке 6 точка
      dP_furnace_7 : Real := -30.0;   // dP в топке 7 точка
      dP_furnace_8 : Real := -30.0;   // dP в топке 8 точка
      P_air_regim_map : Real;   // Р воздуха по режимной карте
      dP_furnace_regim_map : Real;   // dP в топке по режимной карте
      Apply : Bool;   // Применить
      Error : Bool;   // Ошибка
      Reset : Bool;   // Сброс
   END_VAR
BEGIN
END_DATA_BLOCK

DATA_BLOCK "Message"   // DB43
{ S7_Optimized_Access := 'FALSE' }
VERSION : 0.1
   VAR
      OFF_Waiting_btn_ventilation : Bool;   // ОТКЛ. Ожидание нажатия кнопки ВЕНТИЛЯЦИЯ
      OFF_Param_ventilation_not_norm : Bool;   // ОТКЛ. Параметры вентиляции не в норме
      VENTILATION_not_initial_state_gas : Bool;   // ВЕНТИЛЯЦИЯ. Механизмы по газу не переведены в исходное состояние
      VENTILATION_DS_need_dist_mode : Bool;   // ВЕНТИЛЯЦИЯ. Необходимо перевести ДС в дистанционный режим
      VENTILATION_DV_need_dist_mode : Bool;   // ВЕНТИЛЯЦИЯ. Необходимо перевести ДВ в дистанционный режим
      VENTILATION_not_initial_state_air : Bool;   // ВЕНТИЛЯЦИЯ. Механизмы по воздуху не переведены в исходное состояние
      VENTILATION_NAV_not_close : Bool;   // ВЕНТИЛЯЦИЯ. НАВ не закрылись
      VENTILATION_NAD_not_open : Bool;   // ВЕНТИЛЯЦИЯ. НАД не открылись
      VENTILATION_NAV_or_NAD_not_open : Bool;   // ВЕНТИЛЯЦИЯ. НАВ или НАД не открылись
      VENTILATION_DS_not_on : Bool;   // ВЕНТИЛЯЦИЯ. ДС не включился
      VENTILATION_DV_not_on : Bool;   // ВЕНТИЛЯЦИЯ. ДВ не включился
      VENTILATION_run : Bool;   // ВЕНТИЛЯЦИЯ. Идет вентиляция топки
      VENTILATION_not : Bool;   // ВЕНТИЛЯЦИЯ. Нет вентиляции топки
      VENTILATION_alarm : Bool;   // ВЕНТИЛЯЦИЯ. Вентиляция не выполнена
      VENTILATION_ok : Bool;   // ВЕНТИЛЯЦИЯ. Вентиляция успешно проведена
      VENTILATION_Check_param : Bool;   // ВЕНТИЛЯЦИЯ. Проверьте параметры вентиляции
      VENTILATION_NAD_not_open_manual : Bool;   // ВЕНТИЛЯЦИЯ. НАД в местном режиме и не открыты
      VENTILATION_NAV_not_open_manual : Bool;   // ВЕНТИЛЯЦИЯ. НАВ в местном режиме и не открыты
      PRESS_not_initial_state_gas : Bool;   // ОПРЕССОВКА. Механизмы по газу не переведены в исходное состояние
      PRESS_ZRG_not_close : Bool;   // ОПРЕССОВКА. ЗРГ не закрылся
      PRESS_ZDG_not_open : Bool;   // ОПРЕССОВКА. ЗДГ не открылся
      PRESS_P_before_BG_alarm : Bool;   // ОПРЕССОВКА. Давление до БГ не в норме, Устраните неисправность и для продолжения нажмите кн. Розжиг
      PRESS_PZK1_or_KO_untight : Bool;   // ОПРЕССОВКА. ПЗК1 или КО негерметичен
      PRESS_Not_orifice_plate_or_PZK1_untight : Bool;   // ОПРЕССОВКА. Нет дроссельной шайбы или ПЗК1 негерметичен
      PRESS_PZK2_or_KB_untight : Bool;   // ОПРЕССОВКА. ПЗК2 или КБ негерметичен
      TEST_PRESS_ok : Bool;   // ТЕСТОВАЯ ОПРЕССОВКА. Прошла успешно
      IGNITION_Not_flame_igniter : Bool;   // РОЗЖИГ. Нет пламени запальника
      IGNITION_Flame_burner_OK : Bool;   // РОЗЖИГ. Есть пламя горелки
      IGNITION_ZRG_not_close : Bool;   // РОЗЖИГ. ЗРГ не закрыт
      IGNITION_PZK2_not_close : Bool;   // РОЗЖИГ. ПЗК2 не закрыт
      IGNITION_KZ_not_close : Bool;   // РОЗЖИГ. КЗ не закрыт
      IGNITION_KB_not_close : Bool;   // РОЗЖИГ. КБ не закрылся
      IGNITION_PZK1_not_open : Bool;   // РОЗЖИГ. ПЗК1 не открылся
      IGNITION_KZ_not_open : Bool;   // РОЗЖИГ. КЗ не открылся
      IGNITION_not_initial_state_gas : Bool;   // РОЗЖИГ. Механизмы по газу не переведены в исходное состояние
      TEST_IGNITION_ok : Bool;   // ТЕСТОВЫЙ РОЗЖИГ. Прошел успешно
      EMERGENCY_STOP_not_initial_state : Bool;   // ЭКСТРЕННЫЙ ОСТАНОВ. Устройства не переведены в исходное состояние
      ALARM_STOP_not_initial_state_gas : Bool;   // АВАРИЙНЫЙ ОСТАНОВ. Механизмы по газу не переведены в исходное состояние
      PLAN_STOP_not_initial_state_gas : Bool;   // ПЛАНОВЫЙ ОСТАНОВ. Механизмы по газу не переведены в исходное состояние
      STOP_PRESS_P_before_BG_min : Bool;   // ПОСТОСТАНОВОЧНАЯ ОПРЕССОВКА. Давление до БГ низкое
      STOP_PRESS_PZK1_or_KO_untight : Bool;   // ПОСТОСТАНОВОЧНАЯ ОПРЕССОВКА. ПЗК1 или КО негерметичен
      STOP_PRESS_PZK2_or_KB_untight : Bool;   // ПОСТОСТАНОВОЧНАЯ ОПРЕССОВКА. ПЗК2 или КБ негерметичен
      STOP_PRESS_success : Bool;   // ПОСТОСТАНОВОЧНАЯ ОПРЕССОВКА. Успешно проведена
      SHORT_VENTILATION_ok : Bool;   // УКОРОЧЕННАЯ ВЕНТИЛЯЦИЯ. проведена
      VENTILATION_BRU_NAD_need_avto_mode : Bool;   // ВЕНТИЛЯЦИЯ. Необходимо перевести БРУ НАД в автоматический режим
      VENTILATION_BRU_NAV_need_avto_mode : Bool;   // ВЕНТИЛЯЦИЯ. Необходимо перевести БРУ НАВ в автоматический режим
   END_VAR
BEGIN
END_DATA_BLOCK

DATA_BLOCK "Timer"   // DB59
{ S7_Optimized_Access := 'TRUE' }
VERSION : 0.1
   VAR
      alarm_1_IN : Bool;
      alarm_1_Q : Bool;
      alarm_1_PT : Time;
      alarm_2_IN : Bool;
      alarm_2_Q : Bool;
      alarm_2_PT : Time;
      alarm_3_IN : Bool;
      alarm_3_Q : Bool;
      alarm_3_PT : Time;
      alarm_4_IN : Bool;
      alarm_4_Q : Bool;
      alarm_4_PT : Time;
      alarm_5_IN : Bool;
      alarm_5_Q : Bool;
      alarm_5_PT : Time;
      alarm_6_IN : Bool;
      alarm_6_Q : Bool;
      alarm_6_PT : Time;
      alarm_7_IN : Bool;
      alarm_7_Q : Bool;
      alarm_7_PT : Time;
      alarm_8_IN : Bool;
      alarm_8_Q : Bool;
      alarm_8_PT : Time;
      alarm_9_IN : Bool;
      alarm_9_Q : Bool;
      alarm_9_PT : Time;
      alarm_10_IN : Bool;
      alarm_10_Q : Bool;
      alarm_10_PT : Time;
      alarm_11_IN : Bool;
      alarm_11_Q : Bool;
      alarm_11_PT : Time;
      alarm_12_IN : Bool;
      alarm_12_Q : Bool;
      alarm_12_PT : Time;
      alarm_13_IN : Bool;
      alarm_13_Q : Bool;
      alarm_13_PT : Time;
      alarm_14_IN : Bool;
      alarm_14_Q : Bool;
      alarm_14_PT : Time;
      alarm_15_IN : Bool;
      alarm_15_Q : Bool;
      alarm_15_PT : Time;
      alarm_16_IN : Bool;
      alarm_16_Q : Bool;
      alarm_16_PT : Time;
      alarm_17_IN : Bool;
      alarm_17_Q : Bool;
      alarm_17_PT : Time;
      warning_1_IN : Bool;
      warning_1_Q : Bool;
      warning_1_PT : Time;
      warning_2_IN : Bool;
      warning_2_Q : Bool;
      warning_2_PT : Time;
      warning_3_IN : Bool;
      warning_3_Q : Bool;
      warning_3_PT : Time;
      protection_1_IN : Bool;
      protection_1_Q : Bool;
      protection_1_PT : Time;
      protection_2_IN : Bool;
      protection_2_Q : Bool;
      protection_2_PT : Time;
      protection_3_IN : Bool;
      protection_3_Q : Bool;
      protection_3_PT : Time;
      protection_4_IN : Bool;
      protection_4_Q : Bool;
      protection_4_PT : Time;
      protection_5_IN : Bool;
      protection_5_Q : Bool;
      protection_5_PT : Time;
      protection_6_IN : Bool;
      protection_6_Q : Bool;
      protection_6_PT : Time;
      protection_7_IN : Bool;
      protection_7_Q : Bool;
      protection_7_PT : Time;
      protection_8_IN : Bool;
      protection_8_Q : Bool;
      protection_8_PT : Time;
      protection_9_IN : Bool;
      protection_9_Q : Bool;
      protection_9_PT : Time;
      protection_10_IN : Bool;
      protection_10_Q : Bool;
      protection_10_PT : Time;
      protection_11_IN : Bool;
      protection_11_Q : Bool;
      protection_11_PT : Time;
      protection_12_IN : Bool;
      protection_12_Q : Bool;
      protection_12_PT : Time;
      protection_13_IN : Bool;
      protection_13_Q : Bool;
      protection_13_PT : Time;
      protection_14_IN : Bool;
      protection_14_Q : Bool;
      protection_14_PT : Time;
      protection_15_IN : Bool;
      protection_15_Q : Bool;
      protection_15_PT : Time;
      protection_16_IN : Bool;
      protection_16_Q : Bool;
      protection_16_PT : Time;
      protection_17_IN : Bool;
      protection_17_Q : Bool;
      protection_17_PT : Time;
      IGNITION_temp_IN : Bool;
      IGNITION_temp_Q : Bool;
      IGNITION_temp_PT : Time;
      IGNITION_control_flame_IN : Bool;
      IGNITION_control_flame_Q : Bool;
      IGNITION_control_flame_PT : Time;
      PRESS_temp_IN : Bool;
      PRESS_temp_Q : Bool;
      PRESS_temp_PT : Time;
      VENTILATION_temp_IN : Bool;
      VENTILATION_temp_Q : Bool;
      VENTILATION_temp_PT : Time;
      VENTILATION_IN : Bool;
      VENTILATION_R : Bool;
      VENTILATION_Q : Bool;
      VENTILATION_PT : Time;
      MIN_POWER_temp_IN : Bool;
      MIN_POWER_temp_Q : Bool;
      MIN_POWER_temp_PT : Time;
      MIN_POWER_1_IN : Bool;
      MIN_POWER_1_Q : Bool;
      MIN_POWER_1_PT : Time;
      MIN_POWER_2_IN : Bool;
      MIN_POWER_2_Q : Bool;
      MIN_POWER_2_PT : Time;
      HEATING_temp_IN : Bool;
      HEATING_temp_Q : Bool;
      HEATING_temp_PT : Time;
      STOP_PRESS_temp_IN : Bool;
      STOP_PRESS_temp_Q : Bool;
      STOP_PRESS_temp_PT : Time;
      SHORT_VENTILATION_temp_IN : Bool;
      SHORT_VENTILATION_temp_Q : Bool;
      SHORT_VENTILATION_temp_PT : Time;
      EMERGENCY_STOP_temp_IN : Bool;
      EMERGENCY_STOP_temp_Q : Bool;
      EMERGENCY_STOP_temp_PT : Time;
      ALARM_STOP_temp_IN : Bool;
      ALARM_STOP_temp_Q : Bool;
      ALARM_STOP_temp_PT : Time;
      PLAN_STOP_temp_IN : Bool;
      PLAN_STOP_temp_Q : Bool;
      PLAN_STOP_temp_PT : Time;
      RUN_temp_IN : Bool;
      RUN_temp_Q : Bool;
      RUN_temp_PT : LTime;
      close_KZ_IN : Bool;
      close_KZ_Q : Bool;
      close_KZ_PT : Time;
      avto_reset_IVN_IN : Bool;
      avto_reset_IVN_Q : Bool;
      avto_reset_IVN_PT : Time;
      IND_1_IN : Bool;
      IND_1_Q : Bool;
      IND_1_PT : Time;
      IND_2_IN : Bool;
      IND_2_Q : Bool;
      IND_2_PT : Time;
      test_sound_IN : Bool;
      test_sound_Q : Bool;
      test_sound_PT : Time;
      Log_IN : Bool;
      Log_Q : Bool;
   END_VAR
   VAR RETAIN
      Log_PT : Time := T#1s500ms;
   END_VAR
BEGIN
END_DATA_BLOCK

DATA_BLOCK "Syst"   // DB66
{ S7_Optimized_Access := 'TRUE' }
VERSION : 0.1
   VAR
      First_scan_reg_map : Bool := true;
   END_VAR
BEGIN
END_DATA_BLOCK

DATA_BLOCK "Engineering_units"   // DB67
{ S7_Optimized_Access := 'FALSE' }
VERSION : 0.1
   VAR
      pressure_01_EU : Word := 3;
      pressure_02_EU : Word := 3;
      pressure_03_EU : Word := 1;
      pressure_04_EU : Word := 1;
      pressure_05_EU : Word := 1;
      pressure_06_EU : Word := 0;
      pressure_07_EU : Word := 0;
      pressure_08_EU : Word := 1;
      pressure_09_EU : Word := 1;
      pressure_10_EU : Word := 1;
   END_VAR
BEGIN
END_DATA_BLOCK

DATA_BLOCK "TIME_converter_DB"   // DB123
{ S7_Optimized_Access := 'TRUE' }
VERSION : 0.1
// stored: InstanceOfName TIME_converter
"TIME_converter"
BEGIN
END_DATA_BLOCK

DATA_BLOCK "LTIME_converter_DB"   // DB125
{ S7_Optimized_Access := 'TRUE' }
VERSION : 0.1
// stored: InstanceOfName LTIME_converter
"LTIME_converter"
BEGIN
END_DATA_BLOCK

// folder: Control_DB

DATA_BLOCK "Control_ZRG"   // DB6
{ S7_Optimized_Access := 'FALSE' }
VERSION : 0.1
   VAR
      Mode : Bool;   // Режим управления (0-ручной, 1-автоматический)
      Manual_open : Bool;   // Ручное управление. Открыть
      Manual_close : Bool;   // Ручное управление. Закрыть
      Mode_from_PLC : Bool;   // Режим управления от ПЛК(0-ручной, 1-автоматический)
      Manual_open_from_PLC : Bool;   // Ручное управление от ПЛК. Открыть
      Manual_close_from_PLC : Bool;   // Ручное управление от ПЛК. Закрыть
      SP_PID : Real;   // ПИД. Уставка
      DB_PID : Real := 0.5;   // ПИД. Зона нечувствительности
      KP_PID : Real := 0.4;   // ПИД. Кп
      TI_PID : UDInt := 30000;   // ПИД. Ти
      TD_PID : UDInt := 100;   // ПИД. Тд
      FMT_PID : UDInt := 30000;   // ПИД. Время хода исполнительного механизма (мс)
      DT_MIN_PID : UDInt := 200;   // ПИД. Величина минимальной длительности импульса (мс)
      GAP : DInt;   // ПИД. Люфт
   END_VAR
BEGIN
END_DATA_BLOCK

DATA_BLOCK "Control_ZDG"   // DB7
{ S7_Optimized_Access := 'FALSE' }
VERSION : 0.1
   VAR
      Mode : Bool;   // Режим управления (0-ручной, 1-автоматический)
      Manual_open : Bool;   // Ручное управление. Открыть
      Manual_close : Bool;   // Ручное управление. Закрыть
      Manual_stop : Bool;   // Ручное управление. Стоп
      Avto_open : Bool;   // Автоматическое управление. Открыть
      Avto_close : Bool;   // Автоматическое управление. Закрыть
      Avto_stop : Bool;   // Автоматическое управление. Стоп
   END_VAR
BEGIN
END_DATA_BLOCK

DATA_BLOCK "Control_KB"   // DB8
{ S7_Optimized_Access := 'FALSE' }
VERSION : 0.1
   VAR
      Mode : Bool;   // Режим управления (0-ручной, 1-автоматический)
      Manual_close : Bool;   // Ручное управление. Закрыть
      Avto_close : Bool;   // Автоматическое управление. Закрыть
   END_VAR
BEGIN
END_DATA_BLOCK

DATA_BLOCK "Control_KO"   // DB9
{ S7_Optimized_Access := 'FALSE' }
VERSION : 0.1
   VAR
      Mode : Bool;   // Режим управления (0-ручной, 1-автоматический)
      Manual_open : Bool;   // Ручное управление. Открыть
      Avto_open : Bool;   // Автоматическое управление. Открыть
   END_VAR
BEGIN
END_DATA_BLOCK

DATA_BLOCK "Control_KZ"   // DB10
{ S7_Optimized_Access := 'FALSE' }
VERSION : 0.1
   VAR
      Mode : Bool;   // Режим управления (0-ручной, 1-автоматический)
      Manual_open : Bool;   // Ручное управление. Открыть
      Avto_open : Bool;   // Автоматическое управление. Открыть
   END_VAR
BEGIN
END_DATA_BLOCK

DATA_BLOCK "Control_PZK1"   // DB11
{ S7_Optimized_Access := 'FALSE' }
VERSION : 0.1
   VAR
      Mode : Bool;   // Режим управления (0-ручной, 1-автоматический)
      Manual_open : Bool;   // Ручное управление. Открыть
      Avto_open : Bool;   // Автоматическое управление. Открыть
   END_VAR
BEGIN
END_DATA_BLOCK

DATA_BLOCK "Control_PZK2"   // DB12
{ S7_Optimized_Access := 'FALSE' }
VERSION : 0.1
   VAR
      Mode : Bool;   // Режим управления (0-ручной, 1-автоматический)
      Manual_open : Bool;   // Ручное управление. Открыть
      Avto_open : Bool;   // Автоматическое управление. Открыть
   END_VAR
BEGIN
END_DATA_BLOCK

DATA_BLOCK "Control_IVN"   // DB13
{ S7_Optimized_Access := 'FALSE' }
VERSION : 0.1
   VAR
      Mode : Bool;   // Режим управления (0-ручной, 1-автоматический)
      Manual_on : Bool;   // Ручное управление. Включить
      Avto_on : Bool;   // Автоматическое управление. Включить
   END_VAR
BEGIN
END_DATA_BLOCK

DATA_BLOCK "Control_ZDSV_before_boiler"   // DB14
{ S7_Optimized_Access := 'FALSE' }
VERSION : 0.1
   VAR
      Mode : Bool;   // Режим управления (0-ручной, 1-автоматический)
      Manual_open : Bool;   // Ручное управление. Открыть
      Manual_close : Bool;   // Ручное управление. Закрыть
      Manual_stop : Bool;   // Ручное управление. Стоп
      Avto_open : Bool;   // Автоматическое управление. Открыть
      Avto_close : Bool;   // Автоматическое управление. Закрыть
      Avto_stop : Bool;   // Автоматическое управление. Стоп
   END_VAR
BEGIN
END_DATA_BLOCK

DATA_BLOCK "Control_ZDSV_after_boiler"   // DB15
{ S7_Optimized_Access := 'FALSE' }
VERSION : 0.1
   VAR
      Mode : Bool;   // Режим управления (0-ручной, 1-автоматический)
      Manual_open : Bool;   // Ручное управление. Открыть
      Manual_close : Bool;   // Ручное управление. Закрыть
      Manual_stop : Bool;   // Ручное управление. Стоп
      Avto_open : Bool;   // Автоматическое управление. Открыть
      Avto_close : Bool;   // Автоматическое управление. Закрыть
      Avto_stop : Bool;   // Автоматическое управление. Стоп
   END_VAR
BEGIN
END_DATA_BLOCK

DATA_BLOCK "Control_NAV"   // DB16
{ S7_Optimized_Access := 'FALSE' }
VERSION : 0.1
   VAR
      Mode : Bool;   // Режим управления (0-ручной, 1-автоматический)
      Manual_open : Bool;   // Ручное управление. Открыть
      Manual_close : Bool;   // Ручное управление. Закрыть
      Mode_from_PLC : Bool;   // Режим управления от ПЛК(0-ручной, 1-автоматический)
      Manual_open_from_PLC : Bool;   // Ручное управление от ПЛК. Открыть
      Manual_close_from_PLC : Bool;   // Ручное управление от ПЛК. Закрыть
      SP_PID : Real;   // ПИД. Уставка
      DB_PID : Real := 2.0;   // ПИД. Зона нечувствительности
      KP_PID : Real := 1.0;   // ПИД. Кп
      TI_PID : UDInt := 10;   // ПИД. Ти
      TD_PID : UDInt := 0;   // ПИД. Тд
      FMT_PID : UDInt := 27000;   // ПИД. Время хода исполнительного механизма (мс)
      DT_MIN_PID : UDInt := 5;   // ПИД. Величина минимальной длительности импульса (мс)
      GAP : DInt;   // ПИД. Люфт
   END_VAR
BEGIN
END_DATA_BLOCK

DATA_BLOCK "Control_NAD"   // DB17
{ S7_Optimized_Access := 'FALSE' }
VERSION : 0.1
   VAR
      Mode : Bool;   // Режим управления (0-ручной, 1-автоматический)
      Manual_open : Bool;   // Ручное управление. Открыть
      Manual_close : Bool;   // Ручное управление. Закрыть
      Mode_from_PLC : Bool;   // Режим управления от ПЛК(0-ручной, 1-автоматический)
      Manual_open_from_PLC : Bool;   // Ручное управление от ПЛК. Открыть
      Manual_close_from_PLC : Bool;   // Ручное управление от ПЛК. Закрыть
      SP_PID : Real;   // ПИД. Уставка
      DB_PID : Real := 4.0;   // ПИД. Зона нечувствительности
      KP_PID : Real := 0.04;   // ПИД. Кп
      TI_PID : UDInt := 500;   // ПИД. Ти
      TD_PID : UDInt := 0;   // ПИД. Тд
      FMT_PID : UDInt := 33000;   // ПИД. Время хода исполнительного механизма (мс)
      DT_MIN_PID : UDInt := 500;   // ПИД. Величина минимальной длительности импульса (мс)
      GAP : DInt;   // ПИД. Люфт
   END_VAR
BEGIN
END_DATA_BLOCK

DATA_BLOCK "Control_DV"   // DB18
{ S7_Optimized_Access := 'FALSE' }
VERSION : 0.1
   VAR
      Mode : Bool;   // Режим управления (0-ручной, 1-автоматический)
      Manual_Start : Bool;   // Ручное управление. Пуск
      Manual_Stop : Bool;   // Ручное управление. Стоп
      Manual_frequency : Real;   // Ручное управление. Задание частоты
      Avto_Start : Bool;   // Автоматическое управление. Пуск
      Avto_Stop : Bool;   // Автоматическое управление. Стоп
      Mode_from_PLC : Bool;   // Режим управления от ПЛК(0-ручной, 1-автоматический)
      Manual_frequency_from_PLC : Real;   // Ручное управление. Задание частоты
      SP_PID : Real;   // ПИД. Уставка
      DB_PID : Real := 10.0;   // ПИД. Зона нечувствительности
      KP_PID : Real := 0.05;   // ПИД. Кп
      TI_PID : UDInt := 5000;   // ПИД. Ти
      TD_PID : UDInt := 0;   // ПИД. Тд
   END_VAR
BEGIN
END_DATA_BLOCK

DATA_BLOCK "Control_DS"   // DB19
{ S7_Optimized_Access := 'FALSE' }
VERSION : 0.1
   VAR
      Mode : Bool;   // Режим управления (0-ручной, 1-автоматический)
      Manual_Start : Bool;   // Ручное управление. Пуск
      Manual_Stop : Bool;   // Ручное управление. Стоп
      Manual_frequency : Real;   // Ручное управление. Задание частоты
      Avto_Start : Bool;   // Автоматическое управление. Пуск
      Avto_Stop : Bool;   // Автоматическое управление. Стоп
      Mode_from_PLC : Bool;   // Режим управления от ПЛК(0-ручной, 1-автоматический)
      Manual_frequency_from_PLC : Real;   // Ручное управление. Задание частоты
      SP_PID : Real;   // ПИД. Уставка
      DB_PID : Real := 2.0;   // ПИД. Зона нечувствительности
      KP_PID : Real := 0.05;   // ПИД. Кп
      TI_PID : UDInt := 3000;   // ПИД. Ти
      TD_PID : UDInt := 0;   // ПИД. Тд
   END_VAR
BEGIN
END_DATA_BLOCK

// folder: System blocks/Program resources

DATA_BLOCK "Timer_VENTILATION_temp_DB"   // DB5
{ S7_Optimized_Access := 'TRUE' }
AUTHOR : Simatic
FAMILY : IEC
NAME : IEC_TMR
VERSION : 1.0
// stored: InstanceOfName IEC_TIMER
"IEC_TIMER"
BEGIN
END_DATA_BLOCK

DATA_BLOCK "Timer_VENTILATION_DB"   // DB40
{ S7_Optimized_Access := 'TRUE' }
AUTHOR : Simatic
FAMILY : IEC
NAME : IEC_TMR
VERSION : 1.0
// stored: InstanceOfName IEC_TIMER
"IEC_TIMER"
BEGIN
END_DATA_BLOCK

DATA_BLOCK "TON_alarm_1_DB"   // DB41
{ S7_Optimized_Access := 'TRUE' }
AUTHOR : Simatic
FAMILY : IEC
NAME : IEC_TMR
VERSION : 1.0
// stored: InstanceOfName IEC_TIMER
"IEC_TIMER"
BEGIN
END_DATA_BLOCK

DATA_BLOCK "TON_alarm_2_DB"   // DB42
{ S7_Optimized_Access := 'TRUE' }
AUTHOR : Simatic
FAMILY : IEC
NAME : IEC_TMR
VERSION : 1.0
// stored: InstanceOfName IEC_TIMER
"IEC_TIMER"
BEGIN
END_DATA_BLOCK

DATA_BLOCK "Timer_PRESS_temp_DB"   // DB44
{ S7_Optimized_Access := 'TRUE' }
AUTHOR : Simatic
FAMILY : IEC
NAME : IEC_TMR
VERSION : 1.0
// stored: InstanceOfName IEC_TIMER
"IEC_TIMER"
BEGIN
END_DATA_BLOCK

DATA_BLOCK "TON_alarm_3_DB"   // DB45
{ S7_Optimized_Access := 'TRUE' }
AUTHOR : Simatic
FAMILY : IEC
NAME : IEC_TMR
VERSION : 1.0
// stored: InstanceOfName IEC_TIMER
"IEC_TIMER"
BEGIN
END_DATA_BLOCK

DATA_BLOCK "TON_alarm_4_DB"   // DB46
{ S7_Optimized_Access := 'TRUE' }
AUTHOR : Simatic
FAMILY : IEC
NAME : IEC_TMR
VERSION : 1.0
// stored: InstanceOfName IEC_TIMER
"IEC_TIMER"
BEGIN
END_DATA_BLOCK

DATA_BLOCK "TON_avto_reset_IVN_DB"   // DB47
{ S7_Optimized_Access := 'TRUE' }
AUTHOR : Simatic
FAMILY : IEC
NAME : IEC_TMR
VERSION : 1.0
// stored: InstanceOfName IEC_TIMER
"IEC_TIMER"
BEGIN
END_DATA_BLOCK

DATA_BLOCK "Timer_IGNITION_temp_DB"   // DB48
{ S7_Optimized_Access := 'TRUE' }
AUTHOR : Simatic
FAMILY : IEC
NAME : IEC_TMR
VERSION : 1.0
// stored: InstanceOfName IEC_TIMER
"IEC_TIMER"
BEGIN
END_DATA_BLOCK

DATA_BLOCK "Timer_IGNITION_control_flame_DB"   // DB49
{ S7_Optimized_Access := 'TRUE' }
AUTHOR : Simatic
FAMILY : IEC
NAME : IEC_TMR
VERSION : 1.0
// stored: InstanceOfName IEC_TIMER
"IEC_TIMER"
BEGIN
END_DATA_BLOCK

DATA_BLOCK "TON_alarm_5_DB"   // DB50
{ S7_Optimized_Access := 'TRUE' }
AUTHOR : Simatic
FAMILY : IEC
NAME : IEC_TMR
VERSION : 1.0
// stored: InstanceOfName IEC_TIMER
"IEC_TIMER"
BEGIN
END_DATA_BLOCK

DATA_BLOCK "TON_close_KZ_DB"   // DB51
{ S7_Optimized_Access := 'TRUE' }
AUTHOR : Simatic
FAMILY : IEC
NAME : IEC_TMR
VERSION : 1.0
// stored: InstanceOfName IEC_TIMER
"IEC_TIMER"
BEGIN
END_DATA_BLOCK

DATA_BLOCK "TON_alarm_6_DB"   // DB52
{ S7_Optimized_Access := 'TRUE' }
AUTHOR : Simatic
FAMILY : IEC
NAME : IEC_TMR
VERSION : 1.0
// stored: InstanceOfName IEC_TIMER
"IEC_TIMER"
BEGIN
END_DATA_BLOCK

DATA_BLOCK "TON_alarm_7_DB"   // DB53
{ S7_Optimized_Access := 'TRUE' }
AUTHOR : Simatic
FAMILY : IEC
NAME : IEC_TMR
VERSION : 1.0
// stored: InstanceOfName IEC_TIMER
"IEC_TIMER"
BEGIN
END_DATA_BLOCK

DATA_BLOCK "Timer_MIN_POWER_temp_DB"   // DB56
{ S7_Optimized_Access := 'TRUE' }
AUTHOR : Simatic
FAMILY : IEC
NAME : IEC_TMR
VERSION : 1.0
// stored: InstanceOfName IEC_TIMER
"IEC_TIMER"
BEGIN
END_DATA_BLOCK

DATA_BLOCK "Timer_MIN_POWER_1_DB"   // DB57
{ S7_Optimized_Access := 'TRUE' }
AUTHOR : Simatic
FAMILY : IEC
NAME : IEC_TMR
VERSION : 1.0
// stored: InstanceOfName IEC_TIMER
"IEC_TIMER"
BEGIN
END_DATA_BLOCK

DATA_BLOCK "Timer_MIN_POWER_2_DB"   // DB58
{ S7_Optimized_Access := 'TRUE' }
AUTHOR : Simatic
FAMILY : IEC
NAME : IEC_TMR
VERSION : 1.0
// stored: InstanceOfName IEC_TIMER
"IEC_TIMER"
BEGIN
END_DATA_BLOCK

DATA_BLOCK "Timer_HEATING_temp_DB"   // DB60
{ S7_Optimized_Access := 'TRUE' }
AUTHOR : Simatic
FAMILY : IEC
NAME : IEC_TMR
VERSION : 1.0
// stored: InstanceOfName IEC_TIMER
"IEC_TIMER"
BEGIN
END_DATA_BLOCK

DATA_BLOCK "Timer_STOP_PRESS_temp_DB"   // DB61
{ S7_Optimized_Access := 'TRUE' }
AUTHOR : Simatic
FAMILY : IEC
NAME : IEC_TMR
VERSION : 1.0
// stored: InstanceOfName IEC_TIMER
"IEC_TIMER"
BEGIN
END_DATA_BLOCK

DATA_BLOCK "Timer_SHORT_VENTILATION_temp_DB"   // DB62
{ S7_Optimized_Access := 'TRUE' }
AUTHOR : Simatic
FAMILY : IEC
NAME : IEC_TMR
VERSION : 1.0
// stored: InstanceOfName IEC_TIMER
"IEC_TIMER"
BEGIN
END_DATA_BLOCK

DATA_BLOCK "TOF_Log_DB"   // DB65
{ S7_Optimized_Access := 'TRUE' }
AUTHOR : Simatic
FAMILY : IEC
NAME : IEC_TMR
VERSION : 1.0
// stored: InstanceOfName IEC_TIMER
"IEC_TIMER"
BEGIN
END_DATA_BLOCK

DATA_BLOCK "TON_protection_13_DB"   // DB77
{ S7_Optimized_Access := 'TRUE' }
AUTHOR : Simatic
FAMILY : IEC
NAME : IEC_TMR
VERSION : 1.0
// stored: InstanceOfName IEC_TIMER
"IEC_TIMER"
BEGIN
END_DATA_BLOCK

DATA_BLOCK "TON_alarm_8_DB"   // DB82
{ S7_Optimized_Access := 'TRUE' }
AUTHOR : Simatic
FAMILY : IEC
NAME : IEC_TMR
VERSION : 1.0
// stored: InstanceOfName IEC_TIMER
"IEC_TIMER"
BEGIN
END_DATA_BLOCK

DATA_BLOCK "TON_alarm_9_DB"   // DB83
{ S7_Optimized_Access := 'TRUE' }
AUTHOR : Simatic
FAMILY : IEC
NAME : IEC_TMR
VERSION : 1.0
// stored: InstanceOfName IEC_TIMER
"IEC_TIMER"
BEGIN
END_DATA_BLOCK

DATA_BLOCK "TON_alarm_10_DB"   // DB84
{ S7_Optimized_Access := 'TRUE' }
AUTHOR : Simatic
FAMILY : IEC
NAME : IEC_TMR
VERSION : 1.0
// stored: InstanceOfName IEC_TIMER
"IEC_TIMER"
BEGIN
END_DATA_BLOCK

DATA_BLOCK "TON_alarm_11_DB"   // DB85
{ S7_Optimized_Access := 'TRUE' }
AUTHOR : Simatic
FAMILY : IEC
NAME : IEC_TMR
VERSION : 1.0
// stored: InstanceOfName IEC_TIMER
"IEC_TIMER"
BEGIN
END_DATA_BLOCK

DATA_BLOCK "TON_alarm_12_DB"   // DB86
{ S7_Optimized_Access := 'TRUE' }
AUTHOR : Simatic
FAMILY : IEC
NAME : IEC_TMR
VERSION : 1.0
// stored: InstanceOfName IEC_TIMER
"IEC_TIMER"
BEGIN
END_DATA_BLOCK

DATA_BLOCK "TON_alarm_13_DB"   // DB87
{ S7_Optimized_Access := 'TRUE' }
AUTHOR : Simatic
FAMILY : IEC
NAME : IEC_TMR
VERSION : 1.0
// stored: InstanceOfName IEC_TIMER
"IEC_TIMER"
BEGIN
END_DATA_BLOCK

DATA_BLOCK "TON_alarm_14_DB"   // DB88
{ S7_Optimized_Access := 'TRUE' }
AUTHOR : Simatic
FAMILY : IEC
NAME : IEC_TMR
VERSION : 1.0
// stored: InstanceOfName IEC_TIMER
"IEC_TIMER"
BEGIN
END_DATA_BLOCK

DATA_BLOCK "TON_alarm_15_DB"   // DB91
{ S7_Optimized_Access := 'TRUE' }
AUTHOR : Simatic
FAMILY : IEC
NAME : IEC_TMR
VERSION : 1.0
// stored: InstanceOfName IEC_TIMER
"IEC_TIMER"
BEGIN
END_DATA_BLOCK

DATA_BLOCK "TON_alarm_16_DB"   // DB92
{ S7_Optimized_Access := 'TRUE' }
AUTHOR : Simatic
FAMILY : IEC
NAME : IEC_TMR
VERSION : 1.0
// stored: InstanceOfName IEC_TIMER
"IEC_TIMER"
BEGIN
END_DATA_BLOCK

DATA_BLOCK "TON_alarm_17_DB"   // DB93
{ S7_Optimized_Access := 'TRUE' }
AUTHOR : Simatic
FAMILY : IEC
NAME : IEC_TMR
VERSION : 1.0
// stored: InstanceOfName IEC_TIMER
"IEC_TIMER"
BEGIN
END_DATA_BLOCK

DATA_BLOCK "Timer_EMERGENCY_STOP_temp_DB"   // DB96
{ S7_Optimized_Access := 'TRUE' }
AUTHOR : Simatic
FAMILY : IEC
NAME : IEC_TMR
VERSION : 1.0
// stored: InstanceOfName IEC_TIMER
"IEC_TIMER"
BEGIN
END_DATA_BLOCK

